ABB RAPID module: pyramid_without_orientation.mod

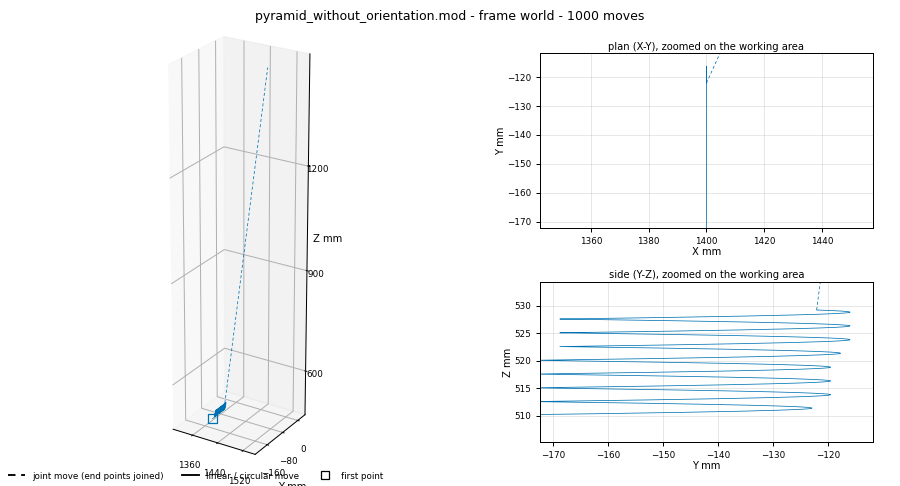
[picture p0: tool path of pyramid_without_orientation.mod in frame world, 1000 of 1000 moves have a stored position in this frame; points joined in program order, loops and branches not executed]
MODULE MainModule
    VAR string program_name:= "ProtoSocketSimulation"; !MODIFIQUE COM O NOME DO PROGRAMA ATUAL!!!!!

    VAR string received_string;
    VAR string message;
    VAR intnum timeint:=0;
    VAR intnum i:=0;
    VAR socketdev socket1;
    VAR string strTemp;
    VAR robtarget actual_pos;
    VAR intnum state;

	TASK PERS tooldata TTW5500_1:=[TRUE,[[32.1099,-0.389434,387.111],[1,0,0,0]],[1,[0,0,100],[1,0,0,0],0,0,0]];
	PERS wobjdata wobj1:=[ FALSE,TRUE,"",[[1400.0000,11.3000,510.0000],[1,0,0,0]],[[0,0,0],[1,0,0,0] ] ];

	CONST robtarget p0:=[[1455.38,0.95,1463.94],[0.707633,-0.000297139,0.70658,0.00010484],[0,0,-1,1],[9E+09,0,0,9E+09,9E+09,9E+09]];
	CONST robtarget p1:=[[0.0000,-194.9500,0.1000],[0.0000,-0.3947,0.9188,0.0000],[-1,0,-1,0],[9E+09,0.0000,0.0000,9E+09,9E+09,9E+09]];
	CONST robtarget p2:=[[0.0000,-193.5108,0.1185],[0.0000,-0.3915,0.9202,0.0000],[-1,0,-1,0],[9E+09,0.0000,-0.4058,9E+09,9E+09,9E+09]];
	CONST robtarget p3:=[[0.0000,-192.0814,0.1370],[0.0000,-0.3882,0.9216,0.0000],[-1,0,-1,0],[9E+09,0.0000,-0.8176,9E+09,9E+09,9E+09]];
	CONST robtarget p4:=[[0.0000,-190.6621,0.1556],[0.0000,-0.3848,0.9230,0.0000],[-1,0,-1,0],[9E+09,0.0000,-1.2355,9E+09,9E+09,9E+09]];
	CONST robtarget p5:=[[0.0000,-189.2531,0.1741],[0.0000,-0.3814,0.9244,0.0000],[-1,0,-1,0],[9E+09,0.0000,-1.6597,9E+09,9E+09,9E+09]];
	CONST robtarget p6:=[[0.0000,-187.8546,0.1926],[0.0000,-0.3779,0.9258,0.0000],[-1,0,-1,0],[9E+09,0.0000,-2.0903,9E+09,9E+09,9E+09]];
	CONST robtarget p7:=[[0.0000,-186.4669,0.2111],[0.0000,-0.3744,0.9273,0.0000],[-1,0,-1,0],[9E+09,0.0000,-2.5273,9E+09,9E+09,9E+09]];
	CONST robtarget p8:=[[0.0000,-185.0902,0.2296],[0.0000,-0.3708,0.9287,0.0000],[-1,0,-1,0],[9E+09,0.0000,-2.9708,9E+09,9E+09,9E+09]];
	CONST robtarget p9:=[[0.0000,-183.7248,0.2481],[0.0000,-0.3671,0.9302,0.0000],[-1,0,-1,0],[9E+09,0.0000,-3.4209,9E+09,9E+09,9E+09]];
	CONST robtarget p10:=[[0.0000,-182.3708,0.2667],[0.0000,-0.3634,0.9316,0.0000],[-1,0,-1,0],[9E+09,0.0000,-3.8777,9E+09,9E+09,9E+09]];
	CONST robtarget p11:=[[0.0000,-181.0287,0.2852],[0.0000,-0.3597,0.9331,0.0000],[-1,0,-1,0],[9E+09,0.0000,-4.3414,9E+09,9E+09,9E+09]];
	CONST robtarget p12:=[[0.0000,-179.6985,0.3037],[0.0000,-0.3558,0.9346,0.0000],[-1,0,-1,0],[9E+09,0.0000,-4.8119,9E+09,9E+09,9E+09]];
	CONST robtarget p13:=[[0.0000,-178.3807,0.3222],[0.0000,-0.3519,0.9360,0.0000],[-1,0,-1,0],[9E+09,0.0000,-5.2895,9E+09,9E+09,9E+09]];
	CONST robtarget p14:=[[0.0000,-177.0755,0.3407],[0.0000,-0.3480,0.9375,0.0000],[-1,0,-1,0],[9E+09,0.0000,-5.7741,9E+09,9E+09,9E+09]];
	CONST robtarget p15:=[[0.0000,-175.7830,0.3593],[0.0000,-0.3439,0.9390,0.0000],[-1,0,-1,0],[9E+09,0.0000,-6.2658,9E+09,9E+09,9E+09]];
	CONST robtarget p16:=[[0.0000,-174.5038,0.3778],[0.0000,-0.3398,0.9405,0.0000],[-1,0,-1,0],[9E+09,0.0000,-6.7648,9E+09,9E+09,9E+09]];
	CONST robtarget p17:=[[0.0000,-173.2379,0.3963],[0.0000,-0.3357,0.9420,0.0000],[-1,0,-1,0],[9E+09,0.0000,-7.2712,9E+09,9E+09,9E+09]];
	CONST robtarget p18:=[[0.0000,-171.9858,0.4148],[0.0000,-0.3315,0.9435,0.0000],[-1,0,-1,0],[9E+09,0.0000,-7.7849,9E+09,9E+09,9E+09]];
	CONST robtarget p19:=[[0.0000,-170.7478,0.4333],[0.0000,-0.3272,0.9450,0.0000],[-1,0,-1,0],[9E+09,0.0000,-8.3062,9E+09,9E+09,9E+09]];
	CONST robtarget p20:=[[0.0000,-169.5240,0.4519],[0.0000,-0.3228,0.9465,0.0000],[-1,0,-1,0],[9E+09,0.0000,-8.8350,9E+09,9E+09,9E+09]];
	CONST robtarget p21:=[[0.0000,-168.3149,0.4704],[0.0000,-0.3184,0.9480,0.0000],[-1,0,-1,0],[9E+09,0.0000,-9.3714,9E+09,9E+09,9E+09]];
	CONST robtarget p22:=[[0.0000,-167.1208,0.4889],[0.0000,-0.3139,0.9495,0.0000],[-1,0,-1,0],[9E+09,0.0000,-9.9156,9E+09,9E+09,9E+09]];
	CONST robtarget p23:=[[0.0000,-165.9420,0.5074],[0.0000,-0.3093,0.9510,0.0000],[-1,0,-1,0],[9E+09,0.0000,-10.4676,9E+09,9E+09,9E+09]];
	CONST robtarget p24:=[[0.0000,-164.7788,0.5259],[0.0000,-0.3046,0.9525,0.0000],[-1,0,-1,0],[9E+09,0.0000,-11.0274,9E+09,9E+09,9E+09]];
	CONST robtarget p25:=[[0.0000,-163.6315,0.5444],[0.0000,-0.2999,0.9540,0.0000],[-1,0,-1,0],[9E+09,0.0000,-11.5951,9E+09,9E+09,9E+09]];
	CONST robtarget p26:=[[0.0000,-162.5006,0.5630],[0.0000,-0.2951,0.9555,0.0000],[-1,0,-1,0],[9E+09,0.0000,-12.1707,9E+09,9E+09,9E+09]];
	CONST robtarget p27:=[[0.0000,-161.3862,0.5815],[0.0000,-0.2902,0.9570,0.0000],[-1,0,-1,0],[9E+09,0.0000,-12.7544,9E+09,9E+09,9E+09]];
	CONST robtarget p28:=[[0.0000,-160.2889,0.6000],[0.0000,-0.2853,0.9584,0.0000],[-1,0,-1,0],[9E+09,0.0000,-13.3461,9E+09,9E+09,9E+09]];
	CONST robtarget p29:=[[0.0000,-159.2088,0.6185],[0.0000,-0.2803,0.9599,0.0000],[-1,0,-1,0],[9E+09,0.0000,-13.9460,9E+09,9E+09,9E+09]];
	CONST robtarget p30:=[[0.0000,-158.1465,0.6370],[0.0000,-0.2752,0.9614,0.0000],[-1,0,-1,0],[9E+09,0.0000,-14.5539,9E+09,9E+09,9E+09]];
	CONST robtarget p31:=[[0.0000,-157.1022,0.6556],[0.0000,-0.2700,0.9629,0.0000],[-1,0,-1,0],[9E+09,0.0000,-15.1700,9E+09,9E+09,9E+09]];
	CONST robtarget p32:=[[0.0000,-156.0763,0.6741],[0.0000,-0.2648,0.9643,0.0000],[-1,0,-1,0],[9E+09,0.0000,-15.7943,9E+09,9E+09,9E+09]];
	CONST robtarget p33:=[[0.0000,-155.0692,0.6926],[0.0000,-0.2594,0.9658,0.0000],[-1,0,-1,0],[9E+09,0.0000,-16.4267,9E+09,9E+09,9E+09]];
	CONST robtarget p34:=[[0.0000,-154.0812,0.7111],[0.0000,-0.2540,0.9672,0.0000],[-1,0,-1,0],[9E+09,0.0000,-17.0674,9E+09,9E+09,9E+09]];
	CONST robtarget p35:=[[0.0000,-153.1128,0.7296],[0.0000,-0.2486,0.9686,0.0000],[-1,0,-1,0],[9E+09,0.0000,-17.7162,9E+09,9E+09,9E+09]];
	CONST robtarget p36:=[[0.0000,-152.1642,0.7481],[0.0000,-0.2430,0.9700,0.0000],[-1,0,-1,0],[9E+09,0.0000,-18.3732,9E+09,9E+09,9E+09]];
	CONST robtarget p37:=[[0.0000,-151.2359,0.7667],[0.0000,-0.2374,0.9714,0.0000],[-1,0,-1,0],[9E+09,0.0000,-19.0384,9E+09,9E+09,9E+09]];
	CONST robtarget p38:=[[0.0000,-150.3282,0.7852],[0.0000,-0.2316,0.9728,0.0000],[-1,0,-1,0],[9E+09,0.0000,-19.7117,9E+09,9E+09,9E+09]];
	CONST robtarget p39:=[[0.0000,-149.4415,0.8037],[0.0000,-0.2259,0.9742,0.0000],[-1,0,-1,0],[9E+09,0.0000,-20.3930,9E+09,9E+09,9E+09]];
	CONST robtarget p40:=[[0.0000,-148.5762,0.8222],[0.0000,-0.2200,0.9755,0.0000],[-1,0,-1,0],[9E+09,0.0000,-21.0824,9E+09,9E+09,9E+09]];
	CONST robtarget p41:=[[0.0000,-147.7327,0.8407],[0.0000,-0.2141,0.9768,0.0000],[-1,0,-1,0],[9E+09,0.0000,-21.7798,9E+09,9E+09,9E+09]];
	CONST robtarget p42:=[[0.0000,-146.9113,0.8593],[0.0000,-0.2080,0.9781,0.0000],[-1,0,-1,0],[9E+09,0.0000,-22.4851,9E+09,9E+09,9E+09]];
	CONST robtarget p43:=[[0.0000,-146.1124,0.8778],[0.0000,-0.2019,0.9794,0.0000],[-1,0,-1,0],[9E+09,0.0000,-23.1982,9E+09,9E+09,9E+09]];
	CONST robtarget p44:=[[0.0000,-145.3364,0.8963],[0.0000,-0.1958,0.9806,0.0000],[-1,0,-1,0],[9E+09,0.0000,-23.9190,9E+09,9E+09,9E+09]];
	CONST robtarget p45:=[[0.0000,-144.5836,0.9148],[0.0000,-0.1895,0.9819,0.0000],[-1,0,-1,0],[9E+09,0.0000,-24.6475,9E+09,9E+09,9E+09]];
	CONST robtarget p46:=[[0.0000,-143.8545,0.9333],[0.0000,-0.1832,0.9831,0.0000],[-1,0,-1,0],[9E+09,0.0000,-25.3834,9E+09,9E+09,9E+09]];
	CONST robtarget p47:=[[0.0000,-143.1493,0.9519],[0.0000,-0.1769,0.9842,0.0000],[-1,0,-1,0],[9E+09,0.0000,-26.1268,9E+09,9E+09,9E+09]];
	CONST robtarget p48:=[[0.0000,-142.4685,0.9704],[0.0000,-0.1704,0.9854,0.0000],[-1,0,-1,0],[9E+09,0.0000,-26.8773,9E+09,9E+09,9E+09]];
	CONST robtarget p49:=[[0.0000,-141.8123,0.9889],[0.0000,-0.1639,0.9865,0.0000],[-1,0,-1,0],[9E+09,0.0000,-27.6350,9E+09,9E+09,9E+09]];
	CONST robtarget p50:=[[0.0000,-141.1812,1.0074],[0.0000,-0.1573,0.9876,0.0000],[-1,0,-1,0],[9E+09,0.0000,-28.3995,9E+09,9E+09,9E+09]];
	CONST robtarget p51:=[[0.0000,-140.5754,1.0259],[0.0000,-0.1507,0.9886,0.0000],[-1,0,-1,0],[9E+09,0.0000,-29.1708,9E+09,9E+09,9E+09]];
	CONST robtarget p52:=[[0.0000,-139.9953,1.0444],[0.0000,-0.1439,0.9896,0.0000],[-1,0,-1,0],[9E+09,0.0000,-29.9486,9E+09,9E+09,9E+09]];
	CONST robtarget p53:=[[0.0000,-139.4412,1.0630],[0.0000,-0.1372,0.9905,0.0000],[-1,0,-1,0],[9E+09,0.0000,-30.7328,9E+09,9E+09,9E+09]];
	CONST robtarget p54:=[[0.0000,-138.9135,1.0815],[0.0000,-0.1303,0.9915,0.0000],[-1,0,-1,0],[9E+09,0.0000,-31.5230,9E+09,9E+09,9E+09]];
	CONST robtarget p55:=[[0.0000,-138.4124,1.1000],[0.0000,-0.1234,0.9924,0.0000],[-1,0,-1,0],[9E+09,0.0000,-32.3191,9E+09,9E+09,9E+09]];
	CONST robtarget p56:=[[0.0000,-137.9381,1.1185],[0.0000,-0.1165,0.9932,0.0000],[-1,0,-1,0],[9E+09,0.0000,-33.1209,9E+09,9E+09,9E+09]];
	CONST robtarget p57:=[[0.0000,-137.4911,1.1370],[0.0000,-0.1095,0.9940,0.0000],[-1,0,-1,0],[9E+09,0.0000,-33.9280,9E+09,9E+09,9E+09]];
	CONST robtarget p58:=[[0.0000,-137.0716,1.1556],[0.0000,-0.1024,0.9947,0.0000],[-1,0,-1,0],[9E+09,0.0000,-34.7402,9E+09,9E+09,9E+09]];
	CONST robtarget p59:=[[0.0000,-136.6797,1.1741],[0.0000,-0.0953,0.9954,0.0000],[-1,0,-1,0],[9E+09,0.0000,-35.5573,9E+09,9E+09,9E+09]];
	CONST robtarget p60:=[[0.0000,-136.3158,1.1926],[0.0000,-0.0882,0.9961,0.0000],[-1,0,-1,0],[9E+09,0.0000,-36.3788,9E+09,9E+09,9E+09]];
	CONST robtarget p61:=[[0.0000,-135.9801,1.2111],[0.0000,-0.0810,0.9967,0.0000],[-1,0,-1,0],[9E+09,0.0000,-37.2046,9E+09,9E+09,9E+09]];
	CONST robtarget p62:=[[0.0000,-135.6728,1.2296],[0.0000,-0.0738,0.9973,0.0000],[-1,0,-1,0],[9E+09,0.0000,-38.0344,9E+09,9E+09,9E+09]];
	CONST robtarget p63:=[[0.0000,-135.3940,1.2481],[0.0000,-0.0666,0.9978,0.0000],[-1,0,-1,0],[9E+09,0.0000,-38.8677,9E+09,9E+09,9E+09]];
	CONST robtarget p64:=[[0.0000,-135.1440,1.2667],[0.0000,-0.0593,0.9982,0.0000],[-1,0,-1,0],[9E+09,0.0000,-39.7042,9E+09,9E+09,9E+09]];
	CONST robtarget p65:=[[0.0000,-134.9229,1.2852],[0.0000,-0.0520,0.9986,0.0000],[-1,0,-1,0],[9E+09,0.0000,-40.5437,9E+09,9E+09,9E+09]];
	CONST robtarget p66:=[[0.0000,-134.7309,1.3037],[0.0000,-0.0446,0.9990,0.0000],[-1,0,-1,0],[9E+09,0.0000,-41.3858,9E+09,9E+09,9E+09]];
	CONST robtarget p67:=[[0.0000,-134.5680,1.3222],[0.0000,-0.0373,0.9993,0.0000],[-1,0,-1,0],[9E+09,0.0000,-42.2301,9E+09,9E+09,9E+09]];
	CONST robtarget p68:=[[0.0000,-134.4344,1.3407],[0.0000,-0.0299,0.9996,0.0000],[-1,0,-1,0],[9E+09,0.0000,-43.0762,9E+09,9E+09,9E+09]];
	CONST robtarget p69:=[[0.0000,-134.3302,1.3593],[0.0000,-0.0225,0.9997,0.0000],[-1,0,-1,0],[9E+09,0.0000,-43.9239,9E+09,9E+09,9E+09]];
	CONST robtarget p70:=[[0.0000,-134.2555,1.3778],[0.0000,-0.0151,0.9999,0.0000],[-1,0,-1,0],[9E+09,0.0000,-44.7727,9E+09,9E+09,9E+09]];
	CONST robtarget p71:=[[0.0000,-134.2102,1.3963],[0.0000,-0.0077,1.0000,0.0000],[-1,0,-1,0],[9E+09,0.0000,-45.6222,9E+09,9E+09,9E+09]];
	CONST robtarget p72:=[[0.0000,-134.1945,1.4148],[0.0000,-0.0002,1.0000,0.0000],[-1,0,-1,0],[9E+09,0.0000,-46.4721,9E+09,9E+09,9E+09]];
	CONST robtarget p73:=[[0.0000,-134.2083,1.4333],[0.0000,-0.0072,-1.0000,0.0000],[-1,0,-1,0],[9E+09,0.0000,-47.3221,9E+09,9E+09,9E+09]];
	CONST robtarget p74:=[[0.0000,-134.2516,1.4519],[0.0000,-0.0146,-0.9999,0.0000],[-1,0,-1,0],[9E+09,0.0000,-48.1716,9E+09,9E+09,9E+09]];
	CONST robtarget p75:=[[0.0000,-134.3244,1.4704],[0.0000,-0.0220,-0.9998,0.0000],[-1,0,-1,0],[9E+09,0.0000,-49.0205,9E+09,9E+09,9E+09]];
	CONST robtarget p76:=[[0.0000,-134.4267,1.4889],[0.0000,-0.0294,-0.9996,0.0000],[-1,0,-1,0],[9E+09,0.0000,-49.8682,9E+09,9E+09,9E+09]];
	CONST robtarget p77:=[[0.0000,-134.5583,1.5074],[0.0000,-0.0368,-0.9993,0.0000],[-1,0,-1,0],[9E+09,0.0000,-50.7145,9E+09,9E+09,9E+09]];
	CONST robtarget p78:=[[0.0000,-134.7192,1.5259],[0.0000,-0.0441,-0.9990,0.0000],[-1,0,-1,0],[9E+09,0.0000,-51.5589,9E+09,9E+09,9E+09]];
	CONST robtarget p79:=[[0.0000,-134.9094,1.5444],[0.0000,-0.0515,-0.9987,0.0000],[-1,0,-1,0],[9E+09,0.0000,-52.4011,9E+09,9E+09,9E+09]];
	CONST robtarget p80:=[[0.0000,-135.1285,1.5630],[0.0000,-0.0588,-0.9983,0.0000],[-1,0,-1,0],[9E+09,0.0000,-53.2408,9E+09,9E+09,9E+09]];
	CONST robtarget p81:=[[0.0000,-135.3767,1.5815],[0.0000,-0.0661,-0.9978,0.0000],[-1,0,-1,0],[9E+09,0.0000,-54.0776,9E+09,9E+09,9E+09]];
	CONST robtarget p82:=[[0.0000,-135.6535,1.6000],[0.0000,-0.0733,-0.9973,0.0000],[-1,0,-1,0],[9E+09,0.0000,-54.9111,9E+09,9E+09,9E+09]];
	CONST robtarget p83:=[[0.0000,-135.9590,1.6185],[0.0000,-0.0806,-0.9968,0.0000],[-1,0,-1,0],[9E+09,0.0000,-55.7411,9E+09,9E+09,9E+09]];
	CONST robtarget p84:=[[0.0000,-136.2929,1.6370],[0.0000,-0.0877,-0.9961,0.0000],[-1,0,-1,0],[9E+09,0.0000,-56.5671,9E+09,9E+09,9E+09]];
	CONST robtarget p85:=[[0.0000,-136.6549,1.6556],[0.0000,-0.0949,-0.9955,0.0000],[-1,0,-1,0],[9E+09,0.0000,-57.3890,9E+09,9E+09,9E+09]];
	CONST robtarget p86:=[[0.0000,-137.0449,1.6741],[0.0000,-0.1020,-0.9948,0.0000],[-1,0,-1,0],[9E+09,0.0000,-58.2064,9E+09,9E+09,9E+09]];
	CONST robtarget p87:=[[0.0000,-137.4627,1.6926],[0.0000,-0.1090,-0.9940,0.0000],[-1,0,-1,0],[9E+09,0.0000,-59.0189,9E+09,9E+09,9E+09]];
	CONST robtarget p88:=[[0.0000,-137.9079,1.7111],[0.0000,-0.1160,-0.9932,0.0000],[-1,0,-1,0],[9E+09,0.0000,-59.8264,9E+09,9E+09,9E+09]];
	CONST robtarget p89:=[[0.0000,-138.3803,1.7296],[0.0000,-0.1230,-0.9924,0.0000],[-1,0,-1,0],[9E+09,0.0000,-60.6285,9E+09,9E+09,9E+09]];
	CONST robtarget p90:=[[0.0000,-138.8797,1.7481],[0.0000,-0.1299,-0.9915,0.0000],[-1,0,-1,0],[9E+09,0.0000,-61.4250,9E+09,9E+09,9E+09]];
	CONST robtarget p91:=[[0.0000,-139.4057,1.7667],[0.0000,-0.1367,-0.9906,0.0000],[-1,0,-1,0],[9E+09,0.0000,-62.2156,9E+09,9E+09,9E+09]];
	CONST robtarget p92:=[[0.0000,-139.9580,1.7852],[0.0000,-0.1435,-0.9897,0.0000],[-1,0,-1,0],[9E+09,0.0000,-63.0002,9E+09,9E+09,9E+09]];
	CONST robtarget p93:=[[0.0000,-140.5364,1.8037],[0.0000,-0.1502,-0.9887,0.0000],[-1,0,-1,0],[9E+09,0.0000,-63.7784,9E+09,9E+09,9E+09]];
	CONST robtarget p94:=[[0.0000,-141.1405,1.8222],[0.0000,-0.1569,-0.9876,0.0000],[-1,0,-1,0],[9E+09,0.0000,-64.5501,9E+09,9E+09,9E+09]];
	CONST robtarget p95:=[[0.0000,-141.7700,1.8407],[0.0000,-0.1635,-0.9866,0.0000],[-1,0,-1,0],[9E+09,0.0000,-65.3151,9E+09,9E+09,9E+09]];
	CONST robtarget p96:=[[0.0000,-142.4245,1.8593],[0.0000,-0.1700,-0.9854,0.0000],[-1,0,-1,0],[9E+09,0.0000,-66.0732,9E+09,9E+09,9E+09]];
	CONST robtarget p97:=[[0.0000,-143.1037,1.8778],[0.0000,-0.1764,-0.9843,0.0000],[-1,0,-1,0],[9E+09,0.0000,-66.8242,9E+09,9E+09,9E+09]];
	CONST robtarget p98:=[[0.0000,-143.8073,1.8963],[0.0000,-0.1828,-0.9831,0.0000],[-1,0,-1,0],[9E+09,0.0000,-67.5681,9E+09,9E+09,9E+09]];
	CONST robtarget p99:=[[0.0000,-144.5349,1.9148],[0.0000,-0.1891,-0.9820,0.0000],[-1,0,-1,0],[9E+09,0.0000,-68.3045,9E+09,9E+09,9E+09]];
	CONST robtarget p100:=[[0.0000,-145.2861,1.9333],[0.0000,-0.1954,-0.9807,0.0000],[-1,0,-1,0],[9E+09,0.0000,-69.0335,9E+09,9E+09,9E+09]];
	CONST robtarget p101:=[[0.0000,-146.0606,1.9519],[0.0000,-0.2015,-0.9795,0.0000],[-1,0,-1,0],[9E+09,0.0000,-69.7548,9E+09,9E+09,9E+09]];
	CONST robtarget p102:=[[0.0000,-146.8580,1.9704],[0.0000,-0.2076,-0.9782,0.0000],[-1,0,-1,0],[9E+09,0.0000,-70.4684,9E+09,9E+09,9E+09]];
	CONST robtarget p103:=[[0.0000,-147.6779,1.9889],[0.0000,-0.2137,-0.9769,0.0000],[-1,0,-1,0],[9E+09,0.0000,-71.1742,9E+09,9E+09,9E+09]];
	CONST robtarget p104:=[[0.0000,-148.5200,2.0074],[0.0000,-0.2196,-0.9756,0.0000],[-1,0,-1,0],[9E+09,0.0000,-71.8721,9E+09,9E+09,9E+09]];
	CONST robtarget p105:=[[0.0000,-149.3839,2.0259],[0.0000,-0.2255,-0.9742,0.0000],[-1,0,-1,0],[9E+09,0.0000,-72.5620,9E+09,9E+09,9E+09]];
	CONST robtarget p106:=[[0.0000,-150.2692,2.0444],[0.0000,-0.2313,-0.9729,0.0000],[-1,0,-1,0],[9E+09,0.0000,-73.2439,9E+09,9E+09,9E+09]];
	CONST robtarget p107:=[[0.0000,-151.1755,2.0630],[0.0000,-0.2370,-0.9715,0.0000],[-1,0,-1,0],[9E+09,0.0000,-73.9178,9E+09,9E+09,9E+09]];
	CONST robtarget p108:=[[0.0000,-152.1025,2.0815],[0.0000,-0.2426,-0.9701,0.0000],[-1,0,-1,0],[9E+09,0.0000,-74.5835,9E+09,9E+09,9E+09]];
	CONST robtarget p109:=[[0.0000,-153.0497,2.1000],[0.0000,-0.2482,-0.9687,0.0000],[-1,0,-1,0],[9E+09,0.0000,-75.2410,9E+09,9E+09,9E+09]];
	CONST robtarget p110:=[[0.0000,-154.0169,2.1185],[0.0000,-0.2537,-0.9673,0.0000],[-1,0,-1,0],[9E+09,0.0000,-75.8904,9E+09,9E+09,9E+09]];
	CONST robtarget p111:=[[0.0000,-155.0036,2.1370],[0.0000,-0.2591,-0.9659,0.0000],[-1,0,-1,0],[9E+09,0.0000,-76.5316,9E+09,9E+09,9E+09]];
	CONST robtarget p112:=[[0.0000,-156.0095,2.1556],[0.0000,-0.2644,-0.9644,0.0000],[-1,0,-1,0],[9E+09,0.0000,-77.1646,9E+09,9E+09,9E+09]];
	CONST robtarget p113:=[[0.0000,-157.0341,2.1741],[0.0000,-0.2697,-0.9630,0.0000],[-1,0,-1,0],[9E+09,0.0000,-77.7894,9E+09,9E+09,9E+09]];
	CONST robtarget p114:=[[0.0000,-158.0772,2.1926],[0.0000,-0.2748,-0.9615,0.0000],[-1,0,-1,0],[9E+09,0.0000,-78.4060,9E+09,9E+09,9E+09]];
	CONST robtarget p115:=[[0.0000,-159.1384,2.2111],[0.0000,-0.2799,-0.9600,0.0000],[-1,0,-1,0],[9E+09,0.0000,-79.0145,9E+09,9E+09,9E+09]];
	CONST robtarget p116:=[[0.0000,-160.2172,2.2296],[0.0000,-0.2850,-0.9585,0.0000],[-1,0,-1,0],[9E+09,0.0000,-79.6148,9E+09,9E+09,9E+09]];
	CONST robtarget p117:=[[0.0000,-161.3135,2.2481],[0.0000,-0.2899,-0.9570,0.0000],[-1,0,-1,0],[9E+09,0.0000,-80.2071,9E+09,9E+09,9E+09]];
	CONST robtarget p118:=[[0.0000,-162.4267,2.2667],[0.0000,-0.2948,-0.9556,0.0000],[-1,0,-1,0],[9E+09,0.0000,-80.7913,9E+09,9E+09,9E+09]];
	CONST robtarget p119:=[[0.0000,-163.5566,2.2852],[0.0000,-0.2996,-0.9541,0.0000],[-1,0,-1,0],[9E+09,0.0000,-81.3675,9E+09,9E+09,9E+09]];
	CONST robtarget p120:=[[0.0000,-164.7028,2.3037],[0.0000,-0.3043,-0.9526,0.0000],[-1,0,-1,0],[9E+09,0.0000,-81.9357,9E+09,9E+09,9E+09]];
	CONST robtarget p121:=[[0.0000,-165.8649,2.3222],[0.0000,-0.3090,-0.9511,0.0000],[-1,0,-1,0],[9E+09,0.0000,-82.4960,9E+09,9E+09,9E+09]];
	CONST robtarget p122:=[[0.0000,-167.0428,2.3407],[0.0000,-0.3136,-0.9496,0.0000],[-1,0,-1,0],[9E+09,0.0000,-83.0485,9E+09,9E+09,9E+09]];
	CONST robtarget p123:=[[0.0000,-168.2359,2.3593],[0.0000,-0.3181,-0.9481,0.0000],[-1,0,-1,0],[9E+09,0.0000,-83.5932,9E+09,9E+09,9E+09]];
	CONST robtarget p124:=[[0.0000,-169.4440,2.3778],[0.0000,-0.3225,-0.9466,0.0000],[-1,0,-1,0],[9E+09,0.0000,-84.1301,9E+09,9E+09,9E+09]];
	CONST robtarget p125:=[[0.0000,-170.6668,2.3963],[0.0000,-0.3269,-0.9451,0.0000],[-1,0,-1,0],[9E+09,0.0000,-84.6595,9E+09,9E+09,9E+09]];
	CONST robtarget p126:=[[0.0000,-171.9039,2.4148],[0.0000,-0.3312,-0.9436,0.0000],[-1,0,-1,0],[9E+09,0.0000,-85.1812,9E+09,9E+09,9E+09]];
	CONST robtarget p127:=[[0.0000,-173.1551,2.4333],[0.0000,-0.3354,-0.9421,0.0000],[-1,0,-1,0],[9E+09,0.0000,-85.6954,9E+09,9E+09,9E+09]];
	CONST robtarget p128:=[[0.0000,-174.4200,2.4519],[0.0000,-0.3396,-0.9406,0.0000],[-1,0,-1,0],[9E+09,0.0000,-86.2023,9E+09,9E+09,9E+09]];
	CONST robtarget p129:=[[0.0000,-175.6984,2.4704],[0.0000,-0.3437,-0.9391,0.0000],[-1,0,-1,0],[9E+09,0.0000,-86.7018,9E+09,9E+09,9E+09]];
	CONST robtarget p130:=[[0.0000,-176.9900,2.4889],[0.0000,-0.3477,-0.9376,0.0000],[-1,0,-1,0],[9E+09,0.0000,-87.1940,9E+09,9E+09,9E+09]];
	CONST robtarget p131:=[[0.0000,-178.2944,2.5074],[0.0000,-0.3517,-0.9361,0.0000],[-1,0,-1,0],[9E+09,0.0000,-87.6791,9E+09,9E+09,9E+09]];
	CONST robtarget p132:=[[0.0000,-179.6114,2.5259],[0.0000,-0.3556,-0.9346,0.0000],[-1,0,-1,0],[9E+09,0.0000,-88.1571,9E+09,9E+09,9E+09]];
	CONST robtarget p133:=[[0.0000,-180.9408,2.5444],[0.0000,-0.3594,-0.9332,0.0000],[-1,0,-1,0],[9E+09,0.0000,-88.6280,9E+09,9E+09,9E+09]];
	CONST robtarget p134:=[[0.0000,-182.2821,2.5630],[0.0000,-0.3632,-0.9317,0.0000],[-1,0,-1,0],[9E+09,0.0000,-89.0921,9E+09,9E+09,9E+09]];
	CONST robtarget p135:=[[0.0000,-183.6353,2.5815],[0.0000,-0.3669,-0.9303,0.0000],[-1,0,-1,0],[9E+09,0.0000,-89.5494,9E+09,9E+09,9E+09]];
	CONST robtarget p136:=[[0.0000,-185.0000,2.6000],[0.0000,-0.3827,0.9239,0.0000],[-1,0,-1,0],[9E+09,0.0000,-90.0000,9E+09,9E+09,9E+09]];
	CONST robtarget p137:=[[0.0000,-183.5932,2.6191],[0.0000,-0.3791,0.9253,0.0000],[-1,0,-1,0],[9E+09,0.0000,-90.4407,9E+09,9E+09,9E+09]];
	CONST robtarget p138:=[[0.0000,-182.1975,2.6382],[0.0000,-0.3755,0.9268,0.0000],[-1,0,-1,0],[9E+09,0.0000,-90.8882,9E+09,9E+09,9E+09]];
	CONST robtarget p139:=[[0.0000,-180.8130,2.6573],[0.0000,-0.3718,0.9283,0.0000],[-1,0,-1,0],[9E+09,0.0000,-91.3426,9E+09,9E+09,9E+09]];
	CONST robtarget p140:=[[0.0000,-179.4401,2.6763],[0.0000,-0.3681,0.9298,0.0000],[-1,0,-1,0],[9E+09,0.0000,-91.8040,9E+09,9E+09,9E+09]];
	CONST robtarget p141:=[[0.0000,-178.0790,2.6954],[0.0000,-0.3643,0.9313,0.0000],[-1,0,-1,0],[9E+09,0.0000,-92.2724,9E+09,9E+09,9E+09]];
	CONST robtarget p142:=[[0.0000,-176.7300,2.7145],[0.0000,-0.3604,0.9328,0.0000],[-1,0,-1,0],[9E+09,0.0000,-92.7481,9E+09,9E+09,9E+09]];
	CONST robtarget p143:=[[0.0000,-175.3933,2.7336],[0.0000,-0.3565,0.9343,0.0000],[-1,0,-1,0],[9E+09,0.0000,-93.2310,9E+09,9E+09,9E+09]];
	CONST robtarget p144:=[[0.0000,-174.0693,2.7527],[0.0000,-0.3525,0.9358,0.0000],[-1,0,-1,0],[9E+09,0.0000,-93.7213,9E+09,9E+09,9E+09]];
	CONST robtarget p145:=[[0.0000,-172.7582,2.7718],[0.0000,-0.3484,0.9373,0.0000],[-1,0,-1,0],[9E+09,0.0000,-94.2191,9E+09,9E+09,9E+09]];
	CONST robtarget p146:=[[0.0000,-171.4604,2.7908],[0.0000,-0.3443,0.9389,0.0000],[-1,0,-1,0],[9E+09,0.0000,-94.7245,9E+09,9E+09,9E+09]];
	CONST robtarget p147:=[[0.0000,-170.1762,2.8099],[0.0000,-0.3401,0.9404,0.0000],[-1,0,-1,0],[9E+09,0.0000,-95.2375,9E+09,9E+09,9E+09]];
	CONST robtarget p148:=[[0.0000,-168.9057,2.8290],[0.0000,-0.3358,0.9419,0.0000],[-1,0,-1,0],[9E+09,0.0000,-95.7583,9E+09,9E+09,9E+09]];
	CONST robtarget p149:=[[0.0000,-167.6495,2.8481],[0.0000,-0.3314,0.9435,0.0000],[-1,0,-1,0],[9E+09,0.0000,-96.2869,9E+09,9E+09,9E+09]];
	CONST robtarget p150:=[[0.0000,-166.4077,2.8672],[0.0000,-0.3270,0.9450,0.0000],[-1,0,-1,0],[9E+09,0.0000,-96.8235,9E+09,9E+09,9E+09]];
	CONST robtarget p151:=[[0.0000,-165.1807,2.8863],[0.0000,-0.3225,0.9466,0.0000],[-1,0,-1,0],[9E+09,0.0000,-97.3681,9E+09,9E+09,9E+09]];
	CONST robtarget p152:=[[0.0000,-163.9689,2.9053],[0.0000,-0.3180,0.9481,0.0000],[-1,0,-1,0],[9E+09,0.0000,-97.9207,9E+09,9E+09,9E+09]];
	CONST robtarget p153:=[[0.0000,-162.7726,2.9244],[0.0000,-0.3133,0.9496,0.0000],[-1,0,-1,0],[9E+09,0.0000,-98.4816,9E+09,9E+09,9E+09]];
	CONST robtarget p154:=[[0.0000,-161.5921,2.9435],[0.0000,-0.3086,0.9512,0.0000],[-1,0,-1,0],[9E+09,0.0000,-99.0507,9E+09,9E+09,9E+09]];
	CONST robtarget p155:=[[0.0000,-160.4277,2.9626],[0.0000,-0.3038,0.9527,0.0000],[-1,0,-1,0],[9E+09,0.0000,-99.6282,9E+09,9E+09,9E+09]];
	CONST robtarget p156:=[[0.0000,-159.2799,2.9817],[0.0000,-0.2989,0.9543,0.0000],[-1,0,-1,0],[9E+09,0.0000,-100.2140,9E+09,9E+09,9E+09]];
	CONST robtarget p157:=[[0.0000,-158.1490,3.0008],[0.0000,-0.2940,0.9558,0.0000],[-1,0,-1,0],[9E+09,0.0000,-100.8082,9E+09,9E+09,9E+09]];
	CONST robtarget p158:=[[0.0000,-157.0354,3.0198],[0.0000,-0.2889,0.9573,0.0000],[-1,0,-1,0],[9E+09,0.0000,-101.4110,9E+09,9E+09,9E+09]];
	CONST robtarget p159:=[[0.0000,-155.9394,3.0389],[0.0000,-0.2838,0.9589,0.0000],[-1,0,-1,0],[9E+09,0.0000,-102.0223,9E+09,9E+09,9E+09]];
	CONST robtarget p160:=[[0.0000,-154.8613,3.0580],[0.0000,-0.2786,0.9604,0.0000],[-1,0,-1,0],[9E+09,0.0000,-102.6422,9E+09,9E+09,9E+09]];
	CONST robtarget p161:=[[0.0000,-153.8017,3.0771],[0.0000,-0.2734,0.9619,0.0000],[-1,0,-1,0],[9E+09,0.0000,-103.2706,9E+09,9E+09,9E+09]];
	CONST robtarget p162:=[[0.0000,-152.7608,3.0962],[0.0000,-0.2680,0.9634,0.0000],[-1,0,-1,0],[9E+09,0.0000,-103.9078,9E+09,9E+09,9E+09]];
	CONST robtarget p163:=[[0.0000,-151.7391,3.1153],[0.0000,-0.2626,0.9649,0.0000],[-1,0,-1,0],[9E+09,0.0000,-104.5536,9E+09,9E+09,9E+09]];
	CONST robtarget p164:=[[0.0000,-150.7369,3.1344],[0.0000,-0.2571,0.9664,0.0000],[-1,0,-1,0],[9E+09,0.0000,-105.2080,9E+09,9E+09,9E+09]];
	CONST robtarget p165:=[[0.0000,-149.7546,3.1534],[0.0000,-0.2515,0.9679,0.0000],[-1,0,-1,0],[9E+09,0.0000,-105.8712,9E+09,9E+09,9E+09]];
	CONST robtarget p166:=[[0.0000,-148.7927,3.1725],[0.0000,-0.2458,0.9693,0.0000],[-1,0,-1,0],[9E+09,0.0000,-106.5430,9E+09,9E+09,9E+09]];
	CONST robtarget p167:=[[0.0000,-147.8514,3.1916],[0.0000,-0.2400,0.9708,0.0000],[-1,0,-1,0],[9E+09,0.0000,-107.2234,9E+09,9E+09,9E+09]];
	CONST robtarget p168:=[[0.0000,-146.9313,3.2107],[0.0000,-0.2342,0.9722,0.0000],[-1,0,-1,0],[9E+09,0.0000,-107.9125,9E+09,9E+09,9E+09]];
	CONST robtarget p169:=[[0.0000,-146.0327,3.2298],[0.0000,-0.2283,0.9736,0.0000],[-1,0,-1,0],[9E+09,0.0000,-108.6102,9E+09,9E+09,9E+09]];
	CONST robtarget p170:=[[0.0000,-145.1561,3.2489],[0.0000,-0.2223,0.9750,0.0000],[-1,0,-1,0],[9E+09,0.0000,-109.3164,9E+09,9E+09,9E+09]];
	CONST robtarget p171:=[[0.0000,-144.3017,3.2679],[0.0000,-0.2162,0.9764,0.0000],[-1,0,-1,0],[9E+09,0.0000,-110.0310,9E+09,9E+09,9E+09]];
	CONST robtarget p172:=[[0.0000,-143.4701,3.2870],[0.0000,-0.2100,0.9777,0.0000],[-1,0,-1,0],[9E+09,0.0000,-110.7541,9E+09,9E+09,9E+09]];
	CONST robtarget p173:=[[0.0000,-142.6615,3.3061],[0.0000,-0.2038,0.9790,0.0000],[-1,0,-1,0],[9E+09,0.0000,-111.4854,9E+09,9E+09,9E+09]];
	CONST robtarget p174:=[[0.0000,-141.8765,3.3252],[0.0000,-0.1974,0.9803,0.0000],[-1,0,-1,0],[9E+09,0.0000,-112.2250,9E+09,9E+09,9E+09]];
	CONST robtarget p175:=[[0.0000,-141.1154,3.3443],[0.0000,-0.1910,0.9816,0.0000],[-1,0,-1,0],[9E+09,0.0000,-112.9727,9E+09,9E+09,9E+09]];
	CONST robtarget p176:=[[0.0000,-140.3786,3.3634],[0.0000,-0.1846,0.9828,0.0000],[-1,0,-1,0],[9E+09,0.0000,-113.7284,9E+09,9E+09,9E+09]];
	CONST robtarget p177:=[[0.0000,-139.6664,3.3824],[0.0000,-0.1780,0.9840,0.0000],[-1,0,-1,0],[9E+09,0.0000,-114.4919,9E+09,9E+09,9E+09]];
	CONST robtarget p178:=[[0.0000,-138.9793,3.4015],[0.0000,-0.1714,0.9852,0.0000],[-1,0,-1,0],[9E+09,0.0000,-115.2631,9E+09,9E+09,9E+09]];
	CONST robtarget p179:=[[0.0000,-138.3177,3.4206],[0.0000,-0.1647,0.9863,0.0000],[-1,0,-1,0],[9E+09,0.0000,-116.0418,9E+09,9E+09,9E+09]];
	CONST robtarget p180:=[[0.0000,-137.6818,3.4397],[0.0000,-0.1579,0.9875,0.0000],[-1,0,-1,0],[9E+09,0.0000,-116.8279,9E+09,9E+09,9E+09]];
	CONST robtarget p181:=[[0.0000,-137.0721,3.4588],[0.0000,-0.1511,0.9885,0.0000],[-1,0,-1,0],[9E+09,0.0000,-117.6211,9E+09,9E+09,9E+09]];
	CONST robtarget p182:=[[0.0000,-136.4888,3.4779],[0.0000,-0.1442,0.9896,0.0000],[-1,0,-1,0],[9E+09,0.0000,-118.4212,9E+09,9E+09,9E+09]];
	CONST robtarget p183:=[[0.0000,-135.9325,3.4969],[0.0000,-0.1372,0.9905,0.0000],[-1,0,-1,0],[9E+09,0.0000,-119.2281,9E+09,9E+09,9E+09]];
	CONST robtarget p184:=[[0.0000,-135.4032,3.5160],[0.0000,-0.1302,0.9915,0.0000],[-1,0,-1,0],[9E+09,0.0000,-120.0414,9E+09,9E+09,9E+09]];
	CONST robtarget p185:=[[0.0000,-134.9015,3.5351],[0.0000,-0.1231,0.9924,0.0000],[-1,0,-1,0],[9E+09,0.0000,-120.8609,9E+09,9E+09,9E+09]];
	CONST robtarget p186:=[[0.0000,-134.4276,3.5542],[0.0000,-0.1159,0.9933,0.0000],[-1,0,-1,0],[9E+09,0.0000,-121.6864,9E+09,9E+09,9E+09]];
	CONST robtarget p187:=[[0.0000,-133.9818,3.5733],[0.0000,-0.1087,0.9941,0.0000],[-1,0,-1,0],[9E+09,0.0000,-122.5175,9E+09,9E+09,9E+09]];
	CONST robtarget p188:=[[0.0000,-133.5644,3.5924],[0.0000,-0.1015,0.9948,0.0000],[-1,0,-1,0],[9E+09,0.0000,-123.3540,9E+09,9E+09,9E+09]];
	CONST robtarget p189:=[[0.0000,-133.1756,3.6115],[0.0000,-0.0941,0.9956,0.0000],[-1,0,-1,0],[9E+09,0.0000,-124.1956,9E+09,9E+09,9E+09]];
	CONST robtarget p190:=[[0.0000,-132.8157,3.6305],[0.0000,-0.0868,0.9962,0.0000],[-1,0,-1,0],[9E+09,0.0000,-125.0419,9E+09,9E+09,9E+09]];
	CONST robtarget p191:=[[0.0000,-132.4849,3.6496],[0.0000,-0.0794,0.9968,0.0000],[-1,0,-1,0],[9E+09,0.0000,-125.8927,9E+09,9E+09,9E+09]];
	CONST robtarget p192:=[[0.0000,-132.1835,3.6687],[0.0000,-0.0720,0.9974,0.0000],[-1,0,-1,0],[9E+09,0.0000,-126.7475,9E+09,9E+09,9E+09]];
	CONST robtarget p193:=[[0.0000,-131.9116,3.6878],[0.0000,-0.0645,0.9979,0.0000],[-1,0,-1,0],[9E+09,0.0000,-127.6060,9E+09,9E+09,9E+09]];
	CONST robtarget p194:=[[0.0000,-131.6695,3.7069],[0.0000,-0.0570,0.9984,0.0000],[-1,0,-1,0],[9E+09,0.0000,-128.4679,9E+09,9E+09,9E+09]];
	CONST robtarget p195:=[[0.0000,-131.4573,3.7260],[0.0000,-0.0494,0.9988,0.0000],[-1,0,-1,0],[9E+09,0.0000,-129.3327,9E+09,9E+09,9E+09]];
	CONST robtarget p196:=[[0.0000,-131.2751,3.7450],[0.0000,-0.0419,0.9991,0.0000],[-1,0,-1,0],[9E+09,0.0000,-130.2002,9E+09,9E+09,9E+09]];
	CONST robtarget p197:=[[0.0000,-131.1231,3.7641],[0.0000,-0.0343,0.9994,0.0000],[-1,0,-1,0],[9E+09,0.0000,-131.0698,9E+09,9E+09,9E+09]];
	CONST robtarget p198:=[[0.0000,-131.0014,3.7832],[0.0000,-0.0267,0.9996,0.0000],[-1,0,-1,0],[9E+09,0.0000,-131.9413,9E+09,9E+09,9E+09]];
	CONST robtarget p199:=[[0.0000,-130.9100,3.8023],[0.0000,-0.0191,0.9998,0.0000],[-1,0,-1,0],[9E+09,0.0000,-132.8142,9E+09,9E+09,9E+09]];
	CONST robtarget p200:=[[0.0000,-130.8491,3.8214],[0.0000,-0.0114,0.9999,0.0000],[-1,0,-1,0],[9E+09,0.0000,-133.6881,9E+09,9E+09,9E+09]];
	CONST robtarget p201:=[[0.0000,-130.8186,3.8405],[0.0000,-0.0038,1.0000,0.0000],[-1,0,-1,0],[9E+09,0.0000,-134.5626,9E+09,9E+09,9E+09]];
	CONST robtarget p202:=[[0.0000,-130.8186,3.8595],[0.0000,-0.0038,-1.0000,0.0000],[-1,0,-1,0],[9E+09,0.0000,-135.4374,9E+09,9E+09,9E+09]];
	CONST robtarget p203:=[[0.0000,-130.8491,3.8786],[0.0000,-0.0114,-0.9999,0.0000],[-1,0,-1,0],[9E+09,0.0000,-136.3119,9E+09,9E+09,9E+09]];
	CONST robtarget p204:=[[0.0000,-130.9100,3.8977],[0.0000,-0.0191,-0.9998,0.0000],[-1,0,-1,0],[9E+09,0.0000,-137.1858,9E+09,9E+09,9E+09]];
	CONST robtarget p205:=[[0.0000,-131.0014,3.9168],[0.0000,-0.0267,-0.9996,0.0000],[-1,0,-1,0],[9E+09,0.0000,-138.0587,9E+09,9E+09,9E+09]];
	CONST robtarget p206:=[[0.0000,-131.1231,3.9359],[0.0000,-0.0343,-0.9994,0.0000],[-1,0,-1,0],[9E+09,0.0000,-138.9302,9E+09,9E+09,9E+09]];
	CONST robtarget p207:=[[0.0000,-131.2751,3.9550],[0.0000,-0.0419,-0.9991,0.0000],[-1,0,-1,0],[9E+09,0.0000,-139.7998,9E+09,9E+09,9E+09]];
	CONST robtarget p208:=[[0.0000,-131.4573,3.9740],[0.0000,-0.0494,-0.9988,0.0000],[-1,0,-1,0],[9E+09,0.0000,-140.6673,9E+09,9E+09,9E+09]];
	CONST robtarget p209:=[[0.0000,-131.6695,3.9931],[0.0000,-0.0570,-0.9984,0.0000],[-1,0,-1,0],[9E+09,0.0000,-141.5321,9E+09,9E+09,9E+09]];
	CONST robtarget p210:=[[0.0000,-131.9116,4.0122],[0.0000,-0.0645,-0.9979,0.0000],[-1,0,-1,0],[9E+09,0.0000,-142.3940,9E+09,9E+09,9E+09]];
	CONST robtarget p211:=[[0.0000,-132.1835,4.0313],[0.0000,-0.0720,-0.9974,0.0000],[-1,0,-1,0],[9E+09,0.0000,-143.2525,9E+09,9E+09,9E+09]];
	CONST robtarget p212:=[[0.0000,-132.4849,4.0504],[0.0000,-0.0794,-0.9968,0.0000],[-1,0,-1,0],[9E+09,0.0000,-144.1073,9E+09,9E+09,9E+09]];
	CONST robtarget p213:=[[0.0000,-132.8157,4.0695],[0.0000,-0.0868,-0.9962,0.0000],[-1,0,-1,0],[9E+09,0.0000,-144.9581,9E+09,9E+09,9E+09]];
	CONST robtarget p214:=[[0.0000,-133.1756,4.0885],[0.0000,-0.0941,-0.9956,0.0000],[-1,0,-1,0],[9E+09,0.0000,-145.8044,9E+09,9E+09,9E+09]];
	CONST robtarget p215:=[[0.0000,-133.5644,4.1076],[0.0000,-0.1015,-0.9948,0.0000],[-1,0,-1,0],[9E+09,0.0000,-146.6460,9E+09,9E+09,9E+09]];
	CONST robtarget p216:=[[0.0000,-133.9818,4.1267],[0.0000,-0.1087,-0.9941,0.0000],[-1,0,-1,0],[9E+09,0.0000,-147.4825,9E+09,9E+09,9E+09]];
	CONST robtarget p217:=[[0.0000,-134.4276,4.1458],[0.0000,-0.1159,-0.9933,0.0000],[-1,0,-1,0],[9E+09,0.0000,-148.3136,9E+09,9E+09,9E+09]];
	CONST robtarget p218:=[[0.0000,-134.9015,4.1649],[0.0000,-0.1231,-0.9924,0.0000],[-1,0,-1,0],[9E+09,0.0000,-149.1391,9E+09,9E+09,9E+09]];
	CONST robtarget p219:=[[0.0000,-135.4032,4.1840],[0.0000,-0.1302,-0.9915,0.0000],[-1,0,-1,0],[9E+09,0.0000,-149.9586,9E+09,9E+09,9E+09]];
	CONST robtarget p220:=[[0.0000,-135.9325,4.2031],[0.0000,-0.1372,-0.9905,0.0000],[-1,0,-1,0],[9E+09,0.0000,-150.7719,9E+09,9E+09,9E+09]];
	CONST robtarget p221:=[[0.0000,-136.4888,4.2221],[0.0000,-0.1442,-0.9896,0.0000],[-1,0,-1,0],[9E+09,0.0000,-151.5788,9E+09,9E+09,9E+09]];
	CONST robtarget p222:=[[0.0000,-137.0721,4.2412],[0.0000,-0.1511,-0.9885,0.0000],[-1,0,-1,0],[9E+09,0.0000,-152.3789,9E+09,9E+09,9E+09]];
	CONST robtarget p223:=[[0.0000,-137.6818,4.2603],[0.0000,-0.1579,-0.9875,0.0000],[-1,0,-1,0],[9E+09,0.0000,-153.1721,9E+09,9E+09,9E+09]];
	CONST robtarget p224:=[[0.0000,-138.3177,4.2794],[0.0000,-0.1647,-0.9863,0.0000],[-1,0,-1,0],[9E+09,0.0000,-153.9582,9E+09,9E+09,9E+09]];
	CONST robtarget p225:=[[0.0000,-138.9793,4.2985],[0.0000,-0.1714,-0.9852,0.0000],[-1,0,-1,0],[9E+09,0.0000,-154.7369,9E+09,9E+09,9E+09]];
	CONST robtarget p226:=[[0.0000,-139.6664,4.3176],[0.0000,-0.1780,-0.9840,0.0000],[-1,0,-1,0],[9E+09,0.0000,-155.5081,9E+09,9E+09,9E+09]];
	CONST robtarget p227:=[[0.0000,-140.3786,4.3366],[0.0000,-0.1846,-0.9828,0.0000],[-1,0,-1,0],[9E+09,0.0000,-156.2716,9E+09,9E+09,9E+09]];
	CONST robtarget p228:=[[0.0000,-141.1154,4.3557],[0.0000,-0.1910,-0.9816,0.0000],[-1,0,-1,0],[9E+09,0.0000,-157.0273,9E+09,9E+09,9E+09]];
	CONST robtarget p229:=[[0.0000,-141.8765,4.3748],[0.0000,-0.1974,-0.9803,0.0000],[-1,0,-1,0],[9E+09,0.0000,-157.7750,9E+09,9E+09,9E+09]];
	CONST robtarget p230:=[[0.0000,-142.6615,4.3939],[0.0000,-0.2038,-0.9790,0.0000],[-1,0,-1,0],[9E+09,0.0000,-158.5146,9E+09,9E+09,9E+09]];
	CONST robtarget p231:=[[0.0000,-143.4701,4.4130],[0.0000,-0.2100,-0.9777,0.0000],[-1,0,-1,0],[9E+09,0.0000,-159.2459,9E+09,9E+09,9E+09]];
	CONST robtarget p232:=[[0.0000,-144.3017,4.4321],[0.0000,-0.2162,-0.9764,0.0000],[-1,0,-1,0],[9E+09,0.0000,-159.9690,9E+09,9E+09,9E+09]];
	CONST robtarget p233:=[[0.0000,-145.1561,4.4511],[0.0000,-0.2223,-0.9750,0.0000],[-1,0,-1,0],[9E+09,0.0000,-160.6836,9E+09,9E+09,9E+09]];
	CONST robtarget p234:=[[0.0000,-146.0327,4.4702],[0.0000,-0.2283,-0.9736,0.0000],[-1,0,-1,0],[9E+09,0.0000,-161.3898,9E+09,9E+09,9E+09]];
	CONST robtarget p235:=[[0.0000,-146.9313,4.4893],[0.0000,-0.2342,-0.9722,0.0000],[-1,0,-1,0],[9E+09,0.0000,-162.0875,9E+09,9E+09,9E+09]];
	CONST robtarget p236:=[[0.0000,-147.8514,4.5084],[0.0000,-0.2400,-0.9708,0.0000],[-1,0,-1,0],[9E+09,0.0000,-162.7766,9E+09,9E+09,9E+09]];
	CONST robtarget p237:=[[0.0000,-148.7927,4.5275],[0.0000,-0.2458,-0.9693,0.0000],[-1,0,-1,0],[9E+09,0.0000,-163.4570,9E+09,9E+09,9E+09]];
	CONST robtarget p238:=[[0.0000,-149.7546,4.5466],[0.0000,-0.2515,-0.9679,0.0000],[-1,0,-1,0],[9E+09,0.0000,-164.1288,9E+09,9E+09,9E+09]];
	CONST robtarget p239:=[[0.0000,-150.7369,4.5656],[0.0000,-0.2571,-0.9664,0.0000],[-1,0,-1,0],[9E+09,0.0000,-164.7920,9E+09,9E+09,9E+09]];
	CONST robtarget p240:=[[0.0000,-151.7391,4.5847],[0.0000,-0.2626,-0.9649,0.0000],[-1,0,-1,0],[9E+09,0.0000,-165.4464,9E+09,9E+09,9E+09]];
	CONST robtarget p241:=[[0.0000,-152.7608,4.6038],[0.0000,-0.2680,-0.9634,0.0000],[-1,0,-1,0],[9E+09,0.0000,-166.0922,9E+09,9E+09,9E+09]];
	CONST robtarget p242:=[[0.0000,-153.8017,4.6229],[0.0000,-0.2734,-0.9619,0.0000],[-1,0,-1,0],[9E+09,0.0000,-166.7294,9E+09,9E+09,9E+09]];
	CONST robtarget p243:=[[0.0000,-154.8613,4.6420],[0.0000,-0.2786,-0.9604,0.0000],[-1,0,-1,0],[9E+09,0.0000,-167.3578,9E+09,9E+09,9E+09]];
	CONST robtarget p244:=[[0.0000,-155.9394,4.6611],[0.0000,-0.2838,-0.9589,0.0000],[-1,0,-1,0],[9E+09,0.0000,-167.9777,9E+09,9E+09,9E+09]];
	CONST robtarget p245:=[[0.0000,-157.0354,4.6802],[0.0000,-0.2889,-0.9573,0.0000],[-1,0,-1,0],[9E+09,0.0000,-168.5890,9E+09,9E+09,9E+09]];
	CONST robtarget p246:=[[0.0000,-158.1490,4.6992],[0.0000,-0.2940,-0.9558,0.0000],[-1,0,-1,0],[9E+09,0.0000,-169.1918,9E+09,9E+09,9E+09]];
	CONST robtarget p247:=[[0.0000,-159.2799,4.7183],[0.0000,-0.2989,-0.9543,0.0000],[-1,0,-1,0],[9E+09,0.0000,-169.7860,9E+09,9E+09,9E+09]];
	CONST robtarget p248:=[[0.0000,-160.4277,4.7374],[0.0000,-0.3038,-0.9527,0.0000],[-1,0,-1,0],[9E+09,0.0000,-170.3718,9E+09,9E+09,9E+09]];
	CONST robtarget p249:=[[0.0000,-161.5921,4.7565],[0.0000,-0.3086,-0.9512,0.0000],[-1,0,-1,0],[9E+09,0.0000,-170.9493,9E+09,9E+09,9E+09]];
	CONST robtarget p250:=[[0.0000,-162.7726,4.7756],[0.0000,-0.3133,-0.9496,0.0000],[-1,0,-1,0],[9E+09,0.0000,-171.5184,9E+09,9E+09,9E+09]];
	CONST robtarget p251:=[[0.0000,-163.9689,4.7947],[0.0000,-0.3180,-0.9481,0.0000],[-1,0,-1,0],[9E+09,0.0000,-172.0793,9E+09,9E+09,9E+09]];
	CONST robtarget p252:=[[0.0000,-165.1807,4.8137],[0.0000,-0.3225,-0.9466,0.0000],[-1,0,-1,0],[9E+09,0.0000,-172.6319,9E+09,9E+09,9E+09]];
	CONST robtarget p253:=[[0.0000,-166.4077,4.8328],[0.0000,-0.3270,-0.9450,0.0000],[-1,0,-1,0],[9E+09,0.0000,-173.1765,9E+09,9E+09,9E+09]];
	CONST robtarget p254:=[[0.0000,-167.6495,4.8519],[0.0000,-0.3314,-0.9435,0.0000],[-1,0,-1,0],[9E+09,0.0000,-173.7131,9E+09,9E+09,9E+09]];
	CONST robtarget p255:=[[0.0000,-168.9057,4.8710],[0.0000,-0.3358,-0.9419,0.0000],[-1,0,-1,0],[9E+09,0.0000,-174.2417,9E+09,9E+09,9E+09]];
	CONST robtarget p256:=[[0.0000,-170.1762,4.8901],[0.0000,-0.3401,-0.9404,0.0000],[-1,0,-1,0],[9E+09,0.0000,-174.7625,9E+09,9E+09,9E+09]];
	CONST robtarget p257:=[[0.0000,-171.4604,4.9092],[0.0000,-0.3443,-0.9389,0.0000],[-1,0,-1,0],[9E+09,0.0000,-175.2755,9E+09,9E+09,9E+09]];
	CONST robtarget p258:=[[0.0000,-172.7582,4.9282],[0.0000,-0.3484,-0.9373,0.0000],[-1,0,-1,0],[9E+09,0.0000,-175.7809,9E+09,9E+09,9E+09]];
	CONST robtarget p259:=[[0.0000,-174.0693,4.9473],[0.0000,-0.3525,-0.9358,0.0000],[-1,0,-1,0],[9E+09,0.0000,-176.2787,9E+09,9E+09,9E+09]];
	CONST robtarget p260:=[[0.0000,-175.3933,4.9664],[0.0000,-0.3565,-0.9343,0.0000],[-1,0,-1,0],[9E+09,0.0000,-176.7690,9E+09,9E+09,9E+09]];
	CONST robtarget p261:=[[0.0000,-176.7300,4.9855],[0.0000,-0.3604,-0.9328,0.0000],[-1,0,-1,0],[9E+09,0.0000,-177.2519,9E+09,9E+09,9E+09]];
	CONST robtarget p262:=[[0.0000,-178.0790,5.0046],[0.0000,-0.3643,-0.9313,0.0000],[-1,0,-1,0],[9E+09,0.0000,-177.7276,9E+09,9E+09,9E+09]];
	CONST robtarget p263:=[[0.0000,-179.4401,5.0237],[0.0000,-0.3681,-0.9298,0.0000],[-1,0,-1,0],[9E+09,0.0000,-178.1960,9E+09,9E+09,9E+09]];
	CONST robtarget p264:=[[0.0000,-180.8130,5.0427],[0.0000,-0.3718,-0.9283,0.0000],[-1,0,-1,0],[9E+09,0.0000,-178.6574,9E+09,9E+09,9E+09]];
	CONST robtarget p265:=[[0.0000,-182.1975,5.0618],[0.0000,-0.3755,-0.9268,0.0000],[-1,0,-1,0],[9E+09,0.0000,-179.1118,9E+09,9E+09,9E+09]];
	CONST robtarget p266:=[[0.0000,-183.5932,5.0809],[0.0000,-0.3791,-0.9253,0.0000],[-1,0,-1,0],[9E+09,0.0000,-179.5593,9E+09,9E+09,9E+09]];
	CONST robtarget p267:=[[0.0000,-185.0000,5.1000],[0.0000,-0.3827,0.9239,0.0000],[-1,0,-1,0],[9E+09,0.0000,-180.0000,9E+09,9E+09,9E+09]];
	CONST robtarget p268:=[[0.0000,-183.5932,5.1191],[0.0000,-0.3791,0.9253,0.0000],[-1,0,-1,0],[9E+09,0.0000,-180.4407,9E+09,9E+09,9E+09]];
	CONST robtarget p269:=[[0.0000,-182.1975,5.1382],[0.0000,-0.3755,0.9268,0.0000],[-1,0,-1,0],[9E+09,0.0000,-180.8882,9E+09,9E+09,9E+09]];
	CONST robtarget p270:=[[0.0000,-180.8130,5.1573],[0.0000,-0.3718,0.9283,0.0000],[-1,0,-1,0],[9E+09,0.0000,-181.3426,9E+09,9E+09,9E+09]];
	CONST robtarget p271:=[[0.0000,-179.4401,5.1763],[0.0000,-0.3681,0.9298,0.0000],[-1,0,-1,0],[9E+09,0.0000,-181.8040,9E+09,9E+09,9E+09]];
	CONST robtarget p272:=[[0.0000,-178.0790,5.1954],[0.0000,-0.3643,0.9313,0.0000],[-1,0,-1,0],[9E+09,0.0000,-182.2724,9E+09,9E+09,9E+09]];
	CONST robtarget p273:=[[0.0000,-176.7300,5.2145],[0.0000,-0.3604,0.9328,0.0000],[-1,0,-1,0],[9E+09,0.0000,-182.7481,9E+09,9E+09,9E+09]];
	CONST robtarget p274:=[[0.0000,-175.3933,5.2336],[0.0000,-0.3565,0.9343,0.0000],[-1,0,-1,0],[9E+09,0.0000,-183.2310,9E+09,9E+09,9E+09]];
	CONST robtarget p275:=[[0.0000,-174.0693,5.2527],[0.0000,-0.3525,0.9358,0.0000],[-1,0,-1,0],[9E+09,0.0000,-183.7213,9E+09,9E+09,9E+09]];
	CONST robtarget p276:=[[0.0000,-172.7582,5.2718],[0.0000,-0.3484,0.9373,0.0000],[-1,0,-1,0],[9E+09,0.0000,-184.2191,9E+09,9E+09,9E+09]];
	CONST robtarget p277:=[[0.0000,-171.4604,5.2908],[0.0000,-0.3443,0.9389,0.0000],[-1,0,-1,0],[9E+09,0.0000,-184.7245,9E+09,9E+09,9E+09]];
	CONST robtarget p278:=[[0.0000,-170.1762,5.3099],[0.0000,-0.3401,0.9404,0.0000],[-1,0,-1,0],[9E+09,0.0000,-185.2375,9E+09,9E+09,9E+09]];
	CONST robtarget p279:=[[0.0000,-168.9057,5.3290],[0.0000,-0.3358,0.9419,0.0000],[-1,0,-1,0],[9E+09,0.0000,-185.7583,9E+09,9E+09,9E+09]];
	CONST robtarget p280:=[[0.0000,-167.6495,5.3481],[0.0000,-0.3314,0.9435,0.0000],[-1,0,-1,0],[9E+09,0.0000,-186.2869,9E+09,9E+09,9E+09]];
	CONST robtarget p281:=[[0.0000,-166.4077,5.3672],[0.0000,-0.3270,0.9450,0.0000],[-1,0,-1,0],[9E+09,0.0000,-186.8235,9E+09,9E+09,9E+09]];
	CONST robtarget p282:=[[0.0000,-165.1807,5.3863],[0.0000,-0.3225,0.9466,0.0000],[-1,0,-1,0],[9E+09,0.0000,-187.3681,9E+09,9E+09,9E+09]];
	CONST robtarget p283:=[[0.0000,-163.9689,5.4053],[0.0000,-0.3180,0.9481,0.0000],[-1,0,-1,0],[9E+09,0.0000,-187.9207,9E+09,9E+09,9E+09]];
	CONST robtarget p284:=[[0.0000,-162.7726,5.4244],[0.0000,-0.3133,0.9496,0.0000],[-1,0,-1,0],[9E+09,0.0000,-188.4816,9E+09,9E+09,9E+09]];
	CONST robtarget p285:=[[0.0000,-161.5921,5.4435],[0.0000,-0.3086,0.9512,0.0000],[-1,0,-1,0],[9E+09,0.0000,-189.0507,9E+09,9E+09,9E+09]];
	CONST robtarget p286:=[[0.0000,-160.4277,5.4626],[0.0000,-0.3038,0.9527,0.0000],[-1,0,-1,0],[9E+09,0.0000,-189.6282,9E+09,9E+09,9E+09]];
	CONST robtarget p287:=[[0.0000,-159.2799,5.4817],[0.0000,-0.2989,0.9543,0.0000],[-1,0,-1,0],[9E+09,0.0000,-190.2140,9E+09,9E+09,9E+09]];
	CONST robtarget p288:=[[0.0000,-158.1490,5.5008],[0.0000,-0.2940,0.9558,0.0000],[-1,0,-1,0],[9E+09,0.0000,-190.8082,9E+09,9E+09,9E+09]];
	CONST robtarget p289:=[[0.0000,-157.0354,5.5198],[0.0000,-0.2889,0.9573,0.0000],[-1,0,-1,0],[9E+09,0.0000,-191.4110,9E+09,9E+09,9E+09]];
	CONST robtarget p290:=[[0.0000,-155.9394,5.5389],[0.0000,-0.2838,0.9589,0.0000],[-1,0,-1,0],[9E+09,0.0000,-192.0223,9E+09,9E+09,9E+09]];
	CONST robtarget p291:=[[0.0000,-154.8613,5.5580],[0.0000,-0.2786,0.9604,0.0000],[-1,0,-1,0],[9E+09,0.0000,-192.6422,9E+09,9E+09,9E+09]];
	CONST robtarget p292:=[[0.0000,-153.8017,5.5771],[0.0000,-0.2734,0.9619,0.0000],[-1,0,-1,0],[9E+09,0.0000,-193.2706,9E+09,9E+09,9E+09]];
	CONST robtarget p293:=[[0.0000,-152.7608,5.5962],[0.0000,-0.2680,0.9634,0.0000],[-1,0,-1,0],[9E+09,0.0000,-193.9078,9E+09,9E+09,9E+09]];
	CONST robtarget p294:=[[0.0000,-151.7391,5.6153],[0.0000,-0.2626,0.9649,0.0000],[-1,0,-1,0],[9E+09,0.0000,-194.5536,9E+09,9E+09,9E+09]];
	CONST robtarget p295:=[[0.0000,-150.7369,5.6344],[0.0000,-0.2571,0.9664,0.0000],[-1,0,-1,0],[9E+09,0.0000,-195.2080,9E+09,9E+09,9E+09]];
	CONST robtarget p296:=[[0.0000,-149.7546,5.6534],[0.0000,-0.2515,0.9679,0.0000],[-1,0,-1,0],[9E+09,0.0000,-195.8712,9E+09,9E+09,9E+09]];
	CONST robtarget p297:=[[0.0000,-148.7927,5.6725],[0.0000,-0.2458,0.9693,0.0000],[-1,0,-1,0],[9E+09,0.0000,-196.5430,9E+09,9E+09,9E+09]];
	CONST robtarget p298:=[[0.0000,-147.8514,5.6916],[0.0000,-0.2400,0.9708,0.0000],[-1,0,-1,0],[9E+09,0.0000,-197.2234,9E+09,9E+09,9E+09]];
	CONST robtarget p299:=[[0.0000,-146.9313,5.7107],[0.0000,-0.2342,0.9722,0.0000],[-1,0,-1,0],[9E+09,0.0000,-197.9125,9E+09,9E+09,9E+09]];
	CONST robtarget p300:=[[0.0000,-146.0327,5.7298],[0.0000,-0.2283,0.9736,0.0000],[-1,0,-1,0],[9E+09,0.0000,-198.6102,9E+09,9E+09,9E+09]];
	CONST robtarget p301:=[[0.0000,-145.1561,5.7489],[0.0000,-0.2223,0.9750,0.0000],[-1,0,-1,0],[9E+09,0.0000,-199.3164,9E+09,9E+09,9E+09]];
	CONST robtarget p302:=[[0.0000,-144.3017,5.7679],[0.0000,-0.2162,0.9764,0.0000],[-1,0,-1,0],[9E+09,0.0000,-200.0310,9E+09,9E+09,9E+09]];
	CONST robtarget p303:=[[0.0000,-143.4701,5.7870],[0.0000,-0.2100,0.9777,0.0000],[-1,0,-1,0],[9E+09,0.0000,-200.7541,9E+09,9E+09,9E+09]];
	CONST robtarget p304:=[[0.0000,-142.6615,5.8061],[0.0000,-0.2038,0.9790,0.0000],[-1,0,-1,0],[9E+09,0.0000,-201.4854,9E+09,9E+09,9E+09]];
	CONST robtarget p305:=[[0.0000,-141.8765,5.8252],[0.0000,-0.1974,0.9803,0.0000],[-1,0,-1,0],[9E+09,0.0000,-202.2250,9E+09,9E+09,9E+09]];
	CONST robtarget p306:=[[0.0000,-141.1154,5.8443],[0.0000,-0.1910,0.9816,0.0000],[-1,0,-1,0],[9E+09,0.0000,-202.9727,9E+09,9E+09,9E+09]];
	CONST robtarget p307:=[[0.0000,-140.3786,5.8634],[0.0000,-0.1846,0.9828,0.0000],[-1,0,-1,0],[9E+09,0.0000,-203.7284,9E+09,9E+09,9E+09]];
	CONST robtarget p308:=[[0.0000,-139.6664,5.8824],[0.0000,-0.1780,0.9840,0.0000],[-1,0,-1,0],[9E+09,0.0000,-204.4919,9E+09,9E+09,9E+09]];
	CONST robtarget p309:=[[0.0000,-138.9793,5.9015],[0.0000,-0.1714,0.9852,0.0000],[-1,0,-1,0],[9E+09,0.0000,-205.2631,9E+09,9E+09,9E+09]];
	CONST robtarget p310:=[[0.0000,-138.3177,5.9206],[0.0000,-0.1647,0.9863,0.0000],[-1,0,-1,0],[9E+09,0.0000,-206.0418,9E+09,9E+09,9E+09]];
	CONST robtarget p311:=[[0.0000,-137.6818,5.9397],[0.0000,-0.1579,0.9875,0.0000],[-1,0,-1,0],[9E+09,0.0000,-206.8279,9E+09,9E+09,9E+09]];
	CONST robtarget p312:=[[0.0000,-137.0721,5.9588],[0.0000,-0.1511,0.9885,0.0000],[-1,0,-1,0],[9E+09,0.0000,-207.6211,9E+09,9E+09,9E+09]];
	CONST robtarget p313:=[[0.0000,-136.4888,5.9779],[0.0000,-0.1442,0.9896,0.0000],[-1,0,-1,0],[9E+09,0.0000,-208.4212,9E+09,9E+09,9E+09]];
	CONST robtarget p314:=[[0.0000,-135.9325,5.9969],[0.0000,-0.1372,0.9905,0.0000],[-1,0,-1,0],[9E+09,0.0000,-209.2281,9E+09,9E+09,9E+09]];
	CONST robtarget p315:=[[0.0000,-135.4032,6.0160],[0.0000,-0.1302,0.9915,0.0000],[-1,0,-1,0],[9E+09,0.0000,-210.0414,9E+09,9E+09,9E+09]];
	CONST robtarget p316:=[[0.0000,-134.9015,6.0351],[0.0000,-0.1231,0.9924,0.0000],[-1,0,-1,0],[9E+09,0.0000,-210.8609,9E+09,9E+09,9E+09]];
	CONST robtarget p317:=[[0.0000,-134.4276,6.0542],[0.0000,-0.1159,0.9933,0.0000],[-1,0,-1,0],[9E+09,0.0000,-211.6864,9E+09,9E+09,9E+09]];
	CONST robtarget p318:=[[0.0000,-133.9818,6.0733],[0.0000,-0.1087,0.9941,0.0000],[-1,0,-1,0],[9E+09,0.0000,-212.5175,9E+09,9E+09,9E+09]];
	CONST robtarget p319:=[[0.0000,-133.5644,6.0924],[0.0000,-0.1015,0.9948,0.0000],[-1,0,-1,0],[9E+09,0.0000,-213.3540,9E+09,9E+09,9E+09]];
	CONST robtarget p320:=[[0.0000,-133.1756,6.1115],[0.0000,-0.0941,0.9956,0.0000],[-1,0,-1,0],[9E+09,0.0000,-214.1956,9E+09,9E+09,9E+09]];
	CONST robtarget p321:=[[0.0000,-132.8157,6.1305],[0.0000,-0.0868,0.9962,0.0000],[-1,0,-1,0],[9E+09,0.0000,-215.0419,9E+09,9E+09,9E+09]];
	CONST robtarget p322:=[[0.0000,-132.4849,6.1496],[0.0000,-0.0794,0.9968,0.0000],[-1,0,-1,0],[9E+09,0.0000,-215.8927,9E+09,9E+09,9E+09]];
	CONST robtarget p323:=[[0.0000,-132.1835,6.1687],[0.0000,-0.0720,0.9974,0.0000],[-1,0,-1,0],[9E+09,0.0000,-216.7475,9E+09,9E+09,9E+09]];
	CONST robtarget p324:=[[0.0000,-131.9116,6.1878],[0.0000,-0.0645,0.9979,0.0000],[-1,0,-1,0],[9E+09,0.0000,-217.6060,9E+09,9E+09,9E+09]];
	CONST robtarget p325:=[[0.0000,-131.6695,6.2069],[0.0000,-0.0570,0.9984,0.0000],[-1,0,-1,0],[9E+09,0.0000,-218.4679,9E+09,9E+09,9E+09]];
	CONST robtarget p326:=[[0.0000,-131.4573,6.2260],[0.0000,-0.0494,0.9988,0.0000],[-1,0,-1,0],[9E+09,0.0000,-219.3327,9E+09,9E+09,9E+09]];
	CONST robtarget p327:=[[0.0000,-131.2751,6.2450],[0.0000,-0.0419,0.9991,0.0000],[-1,0,-1,0],[9E+09,0.0000,-220.2002,9E+09,9E+09,9E+09]];
	CONST robtarget p328:=[[0.0000,-131.1231,6.2641],[0.0000,-0.0343,0.9994,0.0000],[-1,0,-1,0],[9E+09,0.0000,-221.0698,9E+09,9E+09,9E+09]];
	CONST robtarget p329:=[[0.0000,-131.0014,6.2832],[0.0000,-0.0267,0.9996,0.0000],[-1,0,-1,0],[9E+09,0.0000,-221.9413,9E+09,9E+09,9E+09]];
	CONST robtarget p330:=[[0.0000,-130.9100,6.3023],[0.0000,-0.0191,0.9998,0.0000],[-1,0,-1,0],[9E+09,0.0000,-222.8142,9E+09,9E+09,9E+09]];
	CONST robtarget p331:=[[0.0000,-130.8491,6.3214],[0.0000,-0.0114,0.9999,0.0000],[-1,0,-1,0],[9E+09,0.0000,-223.6881,9E+09,9E+09,9E+09]];
	CONST robtarget p332:=[[0.0000,-130.8186,6.3405],[0.0000,-0.0038,1.0000,0.0000],[-1,0,-1,0],[9E+09,0.0000,-224.5626,9E+09,9E+09,9E+09]];
	CONST robtarget p333:=[[0.0000,-130.8186,6.3595],[0.0000,-0.0038,-1.0000,0.0000],[-1,0,-1,0],[9E+09,0.0000,-225.4374,9E+09,9E+09,9E+09]];
	CONST robtarget p334:=[[0.0000,-130.8491,6.3786],[0.0000,-0.0114,-0.9999,0.0000],[-1,0,-1,0],[9E+09,0.0000,-226.3119,9E+09,9E+09,9E+09]];
	CONST robtarget p335:=[[0.0000,-130.9100,6.3977],[0.0000,-0.0191,-0.9998,0.0000],[-1,0,-1,0],[9E+09,0.0000,-227.1858,9E+09,9E+09,9E+09]];
	CONST robtarget p336:=[[0.0000,-131.0014,6.4168],[0.0000,-0.0267,-0.9996,0.0000],[-1,0,-1,0],[9E+09,0.0000,-228.0587,9E+09,9E+09,9E+09]];
	CONST robtarget p337:=[[0.0000,-131.1231,6.4359],[0.0000,-0.0343,-0.9994,0.0000],[-1,0,-1,0],[9E+09,0.0000,-228.9302,9E+09,9E+09,9E+09]];
	CONST robtarget p338:=[[0.0000,-131.2751,6.4550],[0.0000,-0.0419,-0.9991,0.0000],[-1,0,-1,0],[9E+09,0.0000,-229.7998,9E+09,9E+09,9E+09]];
	CONST robtarget p339:=[[0.0000,-131.4573,6.4740],[0.0000,-0.0494,-0.9988,0.0000],[-1,0,-1,0],[9E+09,0.0000,-230.6673,9E+09,9E+09,9E+09]];
	CONST robtarget p340:=[[0.0000,-131.6695,6.4931],[0.0000,-0.0570,-0.9984,0.0000],[-1,0,-1,0],[9E+09,0.0000,-231.5321,9E+09,9E+09,9E+09]];
	CONST robtarget p341:=[[0.0000,-131.9116,6.5122],[0.0000,-0.0645,-0.9979,0.0000],[-1,0,-1,0],[9E+09,0.0000,-232.3940,9E+09,9E+09,9E+09]];
	CONST robtarget p342:=[[0.0000,-132.1835,6.5313],[0.0000,-0.0720,-0.9974,0.0000],[-1,0,-1,0],[9E+09,0.0000,-233.2525,9E+09,9E+09,9E+09]];
	CONST robtarget p343:=[[0.0000,-132.4849,6.5504],[0.0000,-0.0794,-0.9968,0.0000],[-1,0,-1,0],[9E+09,0.0000,-234.1073,9E+09,9E+09,9E+09]];
	CONST robtarget p344:=[[0.0000,-132.8157,6.5695],[0.0000,-0.0868,-0.9962,0.0000],[-1,0,-1,0],[9E+09,0.0000,-234.9581,9E+09,9E+09,9E+09]];
	CONST robtarget p345:=[[0.0000,-133.1756,6.5885],[0.0000,-0.0941,-0.9956,0.0000],[-1,0,-1,0],[9E+09,0.0000,-235.8044,9E+09,9E+09,9E+09]];
	CONST robtarget p346:=[[0.0000,-133.5644,6.6076],[0.0000,-0.1015,-0.9948,0.0000],[-1,0,-1,0],[9E+09,0.0000,-236.6460,9E+09,9E+09,9E+09]];
	CONST robtarget p347:=[[0.0000,-133.9818,6.6267],[0.0000,-0.1087,-0.9941,0.0000],[-1,0,-1,0],[9E+09,0.0000,-237.4825,9E+09,9E+09,9E+09]];
	CONST robtarget p348:=[[0.0000,-134.4276,6.6458],[0.0000,-0.1159,-0.9933,0.0000],[-1,0,-1,0],[9E+09,0.0000,-238.3136,9E+09,9E+09,9E+09]];
	CONST robtarget p349:=[[0.0000,-134.9015,6.6649],[0.0000,-0.1231,-0.9924,0.0000],[-1,0,-1,0],[9E+09,0.0000,-239.1391,9E+09,9E+09,9E+09]];
	CONST robtarget p350:=[[0.0000,-135.4032,6.6840],[0.0000,-0.1302,-0.9915,0.0000],[-1,0,-1,0],[9E+09,0.0000,-239.9586,9E+09,9E+09,9E+09]];
	CONST robtarget p351:=[[0.0000,-135.9325,6.7031],[0.0000,-0.1372,-0.9905,0.0000],[-1,0,-1,0],[9E+09,0.0000,-240.7719,9E+09,9E+09,9E+09]];
	CONST robtarget p352:=[[0.0000,-136.4888,6.7221],[0.0000,-0.1442,-0.9896,0.0000],[-1,0,-1,0],[9E+09,0.0000,-241.5788,9E+09,9E+09,9E+09]];
	CONST robtarget p353:=[[0.0000,-137.0721,6.7412],[0.0000,-0.1511,-0.9885,0.0000],[-1,0,-1,0],[9E+09,0.0000,-242.3789,9E+09,9E+09,9E+09]];
	CONST robtarget p354:=[[0.0000,-137.6818,6.7603],[0.0000,-0.1579,-0.9875,0.0000],[-1,0,-1,0],[9E+09,0.0000,-243.1721,9E+09,9E+09,9E+09]];
	CONST robtarget p355:=[[0.0000,-138.3177,6.7794],[0.0000,-0.1647,-0.9863,0.0000],[-1,0,-1,0],[9E+09,0.0000,-243.9582,9E+09,9E+09,9E+09]];
	CONST robtarget p356:=[[0.0000,-138.9793,6.7985],[0.0000,-0.1714,-0.9852,0.0000],[-1,0,-1,0],[9E+09,0.0000,-244.7369,9E+09,9E+09,9E+09]];
	CONST robtarget p357:=[[0.0000,-139.6664,6.8176],[0.0000,-0.1780,-0.9840,0.0000],[-1,0,-1,0],[9E+09,0.0000,-245.5081,9E+09,9E+09,9E+09]];
	CONST robtarget p358:=[[0.0000,-140.3786,6.8366],[0.0000,-0.1846,-0.9828,0.0000],[-1,0,-1,0],[9E+09,0.0000,-246.2716,9E+09,9E+09,9E+09]];
	CONST robtarget p359:=[[0.0000,-141.1154,6.8557],[0.0000,-0.1910,-0.9816,0.0000],[-1,0,-1,0],[9E+09,0.0000,-247.0273,9E+09,9E+09,9E+09]];
	CONST robtarget p360:=[[0.0000,-141.8765,6.8748],[0.0000,-0.1974,-0.9803,0.0000],[-1,0,-1,0],[9E+09,0.0000,-247.7750,9E+09,9E+09,9E+09]];
	CONST robtarget p361:=[[0.0000,-142.6615,6.8939],[0.0000,-0.2038,-0.9790,0.0000],[-1,0,-1,0],[9E+09,0.0000,-248.5146,9E+09,9E+09,9E+09]];
	CONST robtarget p362:=[[0.0000,-143.4701,6.9130],[0.0000,-0.2100,-0.9777,0.0000],[-1,0,-1,0],[9E+09,0.0000,-249.2459,9E+09,9E+09,9E+09]];
	CONST robtarget p363:=[[0.0000,-144.3017,6.9321],[0.0000,-0.2162,-0.9764,0.0000],[-1,0,-1,0],[9E+09,0.0000,-249.9690,9E+09,9E+09,9E+09]];
	CONST robtarget p364:=[[0.0000,-145.1561,6.9511],[0.0000,-0.2223,-0.9750,0.0000],[-1,0,-1,0],[9E+09,0.0000,-250.6836,9E+09,9E+09,9E+09]];
	CONST robtarget p365:=[[0.0000,-146.0327,6.9702],[0.0000,-0.2283,-0.9736,0.0000],[-1,0,-1,0],[9E+09,0.0000,-251.3898,9E+09,9E+09,9E+09]];
	CONST robtarget p366:=[[0.0000,-146.9313,6.9893],[0.0000,-0.2342,-0.9722,0.0000],[-1,0,-1,0],[9E+09,0.0000,-252.0875,9E+09,9E+09,9E+09]];
	CONST robtarget p367:=[[0.0000,-147.8514,7.0084],[0.0000,-0.2400,-0.9708,0.0000],[-1,0,-1,0],[9E+09,0.0000,-252.7766,9E+09,9E+09,9E+09]];
	CONST robtarget p368:=[[0.0000,-148.7927,7.0275],[0.0000,-0.2458,-0.9693,0.0000],[-1,0,-1,0],[9E+09,0.0000,-253.4570,9E+09,9E+09,9E+09]];
	CONST robtarget p369:=[[0.0000,-149.7546,7.0466],[0.0000,-0.2515,-0.9679,0.0000],[-1,0,-1,0],[9E+09,0.0000,-254.1288,9E+09,9E+09,9E+09]];
	CONST robtarget p370:=[[0.0000,-150.7369,7.0656],[0.0000,-0.2571,-0.9664,0.0000],[-1,0,-1,0],[9E+09,0.0000,-254.7920,9E+09,9E+09,9E+09]];
	CONST robtarget p371:=[[0.0000,-151.7391,7.0847],[0.0000,-0.2626,-0.9649,0.0000],[-1,0,-1,0],[9E+09,0.0000,-255.4464,9E+09,9E+09,9E+09]];
	CONST robtarget p372:=[[0.0000,-152.7608,7.1038],[0.0000,-0.2680,-0.9634,0.0000],[-1,0,-1,0],[9E+09,0.0000,-256.0922,9E+09,9E+09,9E+09]];
	CONST robtarget p373:=[[0.0000,-153.8017,7.1229],[0.0000,-0.2734,-0.9619,0.0000],[-1,0,-1,0],[9E+09,0.0000,-256.7294,9E+09,9E+09,9E+09]];
	CONST robtarget p374:=[[0.0000,-154.8613,7.1420],[0.0000,-0.2786,-0.9604,0.0000],[-1,0,-1,0],[9E+09,0.0000,-257.3578,9E+09,9E+09,9E+09]];
	CONST robtarget p375:=[[0.0000,-155.9394,7.1611],[0.0000,-0.2838,-0.9589,0.0000],[-1,0,-1,0],[9E+09,0.0000,-257.9777,9E+09,9E+09,9E+09]];
	CONST robtarget p376:=[[0.0000,-157.0354,7.1802],[0.0000,-0.2889,-0.9573,0.0000],[-1,0,-1,0],[9E+09,0.0000,-258.5890,9E+09,9E+09,9E+09]];
	CONST robtarget p377:=[[0.0000,-158.1490,7.1992],[0.0000,-0.2940,-0.9558,0.0000],[-1,0,-1,0],[9E+09,0.0000,-259.1918,9E+09,9E+09,9E+09]];
	CONST robtarget p378:=[[0.0000,-159.2799,7.2183],[0.0000,-0.2989,-0.9543,0.0000],[-1,0,-1,0],[9E+09,0.0000,-259.7860,9E+09,9E+09,9E+09]];
	CONST robtarget p379:=[[0.0000,-160.4277,7.2374],[0.0000,-0.3038,-0.9527,0.0000],[-1,0,-1,0],[9E+09,0.0000,-260.3718,9E+09,9E+09,9E+09]];
	CONST robtarget p380:=[[0.0000,-161.5921,7.2565],[0.0000,-0.3086,-0.9512,0.0000],[-1,0,-1,0],[9E+09,0.0000,-260.9493,9E+09,9E+09,9E+09]];
	CONST robtarget p381:=[[0.0000,-162.7726,7.2756],[0.0000,-0.3133,-0.9496,0.0000],[-1,0,-1,0],[9E+09,0.0000,-261.5184,9E+09,9E+09,9E+09]];
	CONST robtarget p382:=[[0.0000,-163.9689,7.2947],[0.0000,-0.3180,-0.9481,0.0000],[-1,0,-1,0],[9E+09,0.0000,-262.0793,9E+09,9E+09,9E+09]];
	CONST robtarget p383:=[[0.0000,-165.1807,7.3137],[0.0000,-0.3225,-0.9466,0.0000],[-1,0,-1,0],[9E+09,0.0000,-262.6319,9E+09,9E+09,9E+09]];
	CONST robtarget p384:=[[0.0000,-166.4077,7.3328],[0.0000,-0.3270,-0.9450,0.0000],[-1,0,-1,0],[9E+09,0.0000,-263.1765,9E+09,9E+09,9E+09]];
	CONST robtarget p385:=[[0.0000,-167.6495,7.3519],[0.0000,-0.3314,-0.9435,0.0000],[-1,0,-1,0],[9E+09,0.0000,-263.7131,9E+09,9E+09,9E+09]];
	CONST robtarget p386:=[[0.0000,-168.9057,7.3710],[0.0000,-0.3358,-0.9419,0.0000],[-1,0,-1,0],[9E+09,0.0000,-264.2417,9E+09,9E+09,9E+09]];
	CONST robtarget p387:=[[0.0000,-170.1762,7.3901],[0.0000,-0.3401,-0.9404,0.0000],[-1,0,-1,0],[9E+09,0.0000,-264.7625,9E+09,9E+09,9E+09]];
	CONST robtarget p388:=[[0.0000,-171.4604,7.4092],[0.0000,-0.3443,-0.9389,0.0000],[-1,0,-1,0],[9E+09,0.0000,-265.2755,9E+09,9E+09,9E+09]];
	CONST robtarget p389:=[[0.0000,-172.7582,7.4282],[0.0000,-0.3484,-0.9373,0.0000],[-1,0,-1,0],[9E+09,0.0000,-265.7809,9E+09,9E+09,9E+09]];
	CONST robtarget p390:=[[0.0000,-174.0693,7.4473],[0.0000,-0.3525,-0.9358,0.0000],[-1,0,-1,0],[9E+09,0.0000,-266.2787,9E+09,9E+09,9E+09]];
	CONST robtarget p391:=[[0.0000,-175.3933,7.4664],[0.0000,-0.3565,-0.9343,0.0000],[-1,0,-1,0],[9E+09,0.0000,-266.7690,9E+09,9E+09,9E+09]];
	CONST robtarget p392:=[[0.0000,-176.7300,7.4855],[0.0000,-0.3604,-0.9328,0.0000],[-1,0,-1,0],[9E+09,0.0000,-267.2519,9E+09,9E+09,9E+09]];
	CONST robtarget p393:=[[0.0000,-178.0790,7.5046],[0.0000,-0.3643,-0.9313,0.0000],[-1,0,-1,0],[9E+09,0.0000,-267.7276,9E+09,9E+09,9E+09]];
	CONST robtarget p394:=[[0.0000,-179.4401,7.5237],[0.0000,-0.3681,-0.9298,0.0000],[-1,0,-1,0],[9E+09,0.0000,-268.1960,9E+09,9E+09,9E+09]];
	CONST robtarget p395:=[[0.0000,-180.8130,7.5427],[0.0000,-0.3718,-0.9283,0.0000],[-1,0,-1,0],[9E+09,0.0000,-268.6574,9E+09,9E+09,9E+09]];
	CONST robtarget p396:=[[0.0000,-182.1975,7.5618],[0.0000,-0.3755,-0.9268,0.0000],[-1,0,-1,0],[9E+09,0.0000,-269.1118,9E+09,9E+09,9E+09]];
	CONST robtarget p397:=[[0.0000,-183.5932,7.5809],[0.0000,-0.3791,-0.9253,0.0000],[-1,0,-1,0],[9E+09,0.0000,-269.5593,9E+09,9E+09,9E+09]];
	CONST robtarget p398:=[[0.0000,-185.0000,7.6000],[0.0000,-0.3827,0.9239,0.0000],[-1,0,-1,0],[9E+09,0.0000,-270.0000,9E+09,9E+09,9E+09]];
	CONST robtarget p399:=[[0.0000,-183.5932,7.6191],[0.0000,-0.3791,0.9253,0.0000],[-1,0,-1,0],[9E+09,0.0000,-270.4407,9E+09,9E+09,9E+09]];
	CONST robtarget p400:=[[0.0000,-182.1975,7.6382],[0.0000,-0.3755,0.9268,0.0000],[-1,0,-1,0],[9E+09,0.0000,-270.8882,9E+09,9E+09,9E+09]];
	CONST robtarget p401:=[[0.0000,-180.8130,7.6573],[0.0000,-0.3718,0.9283,0.0000],[-1,0,-1,0],[9E+09,0.0000,-271.3426,9E+09,9E+09,9E+09]];
	CONST robtarget p402:=[[0.0000,-179.4401,7.6763],[0.0000,-0.3681,0.9298,0.0000],[-1,0,-1,0],[9E+09,0.0000,-271.8040,9E+09,9E+09,9E+09]];
	CONST robtarget p403:=[[0.0000,-178.0790,7.6954],[0.0000,-0.3643,0.9313,0.0000],[-1,0,-1,0],[9E+09,0.0000,-272.2724,9E+09,9E+09,9E+09]];
	CONST robtarget p404:=[[0.0000,-176.7300,7.7145],[0.0000,-0.3604,0.9328,0.0000],[-1,0,-1,0],[9E+09,0.0000,-272.7481,9E+09,9E+09,9E+09]];
	CONST robtarget p405:=[[0.0000,-175.3933,7.7336],[0.0000,-0.3565,0.9343,0.0000],[-1,0,-1,0],[9E+09,0.0000,-273.2310,9E+09,9E+09,9E+09]];
	CONST robtarget p406:=[[0.0000,-174.0693,7.7527],[0.0000,-0.3525,0.9358,0.0000],[-1,0,-1,0],[9E+09,0.0000,-273.7213,9E+09,9E+09,9E+09]];
	CONST robtarget p407:=[[0.0000,-172.7582,7.7718],[0.0000,-0.3484,0.9373,0.0000],[-1,0,-1,0],[9E+09,0.0000,-274.2191,9E+09,9E+09,9E+09]];
	CONST robtarget p408:=[[0.0000,-171.4604,7.7908],[0.0000,-0.3443,0.9389,0.0000],[-1,0,-1,0],[9E+09,0.0000,-274.7245,9E+09,9E+09,9E+09]];
	CONST robtarget p409:=[[0.0000,-170.1762,7.8099],[0.0000,-0.3401,0.9404,0.0000],[-1,0,-1,0],[9E+09,0.0000,-275.2375,9E+09,9E+09,9E+09]];
	CONST robtarget p410:=[[0.0000,-168.9057,7.8290],[0.0000,-0.3358,0.9419,0.0000],[-1,0,-1,0],[9E+09,0.0000,-275.7583,9E+09,9E+09,9E+09]];
	CONST robtarget p411:=[[0.0000,-167.6495,7.8481],[0.0000,-0.3314,0.9435,0.0000],[-1,0,-1,0],[9E+09,0.0000,-276.2869,9E+09,9E+09,9E+09]];
	CONST robtarget p412:=[[0.0000,-166.4077,7.8672],[0.0000,-0.3270,0.9450,0.0000],[-1,0,-1,0],[9E+09,0.0000,-276.8235,9E+09,9E+09,9E+09]];
	CONST robtarget p413:=[[0.0000,-165.1807,7.8863],[0.0000,-0.3225,0.9466,0.0000],[-1,0,-1,0],[9E+09,0.0000,-277.3681,9E+09,9E+09,9E+09]];
	CONST robtarget p414:=[[0.0000,-163.9689,7.9053],[0.0000,-0.3180,0.9481,0.0000],[-1,0,-1,0],[9E+09,0.0000,-277.9207,9E+09,9E+09,9E+09]];
	CONST robtarget p415:=[[0.0000,-162.7726,7.9244],[0.0000,-0.3133,0.9496,0.0000],[-1,0,-1,0],[9E+09,0.0000,-278.4816,9E+09,9E+09,9E+09]];
	CONST robtarget p416:=[[0.0000,-161.5921,7.9435],[0.0000,-0.3086,0.9512,0.0000],[-1,0,-1,0],[9E+09,0.0000,-279.0507,9E+09,9E+09,9E+09]];
	CONST robtarget p417:=[[0.0000,-160.4277,7.9626],[0.0000,-0.3038,0.9527,0.0000],[-1,0,-1,0],[9E+09,0.0000,-279.6282,9E+09,9E+09,9E+09]];
	CONST robtarget p418:=[[0.0000,-159.2799,7.9817],[0.0000,-0.2989,0.9543,0.0000],[-1,0,-1,0],[9E+09,0.0000,-280.2140,9E+09,9E+09,9E+09]];
	CONST robtarget p419:=[[0.0000,-158.1490,8.0008],[0.0000,-0.2940,0.9558,0.0000],[-1,0,-1,0],[9E+09,0.0000,-280.8082,9E+09,9E+09,9E+09]];
	CONST robtarget p420:=[[0.0000,-157.0354,8.0198],[0.0000,-0.2889,0.9573,0.0000],[-1,0,-1,0],[9E+09,0.0000,-281.4110,9E+09,9E+09,9E+09]];
	CONST robtarget p421:=[[0.0000,-155.9394,8.0389],[0.0000,-0.2838,0.9589,0.0000],[-1,0,-1,0],[9E+09,0.0000,-282.0223,9E+09,9E+09,9E+09]];
	CONST robtarget p422:=[[0.0000,-154.8613,8.0580],[0.0000,-0.2786,0.9604,0.0000],[-1,0,-1,0],[9E+09,0.0000,-282.6422,9E+09,9E+09,9E+09]];
	CONST robtarget p423:=[[0.0000,-153.8017,8.0771],[0.0000,-0.2734,0.9619,0.0000],[-1,0,-1,0],[9E+09,0.0000,-283.2706,9E+09,9E+09,9E+09]];
	CONST robtarget p424:=[[0.0000,-152.7608,8.0962],[0.0000,-0.2680,0.9634,0.0000],[-1,0,-1,0],[9E+09,0.0000,-283.9078,9E+09,9E+09,9E+09]];
	CONST robtarget p425:=[[0.0000,-151.7391,8.1153],[0.0000,-0.2626,0.9649,0.0000],[-1,0,-1,0],[9E+09,0.0000,-284.5536,9E+09,9E+09,9E+09]];
	CONST robtarget p426:=[[0.0000,-150.7369,8.1344],[0.0000,-0.2571,0.9664,0.0000],[-1,0,-1,0],[9E+09,0.0000,-285.2080,9E+09,9E+09,9E+09]];
	CONST robtarget p427:=[[0.0000,-149.7546,8.1534],[0.0000,-0.2515,0.9679,0.0000],[-1,0,-1,0],[9E+09,0.0000,-285.8712,9E+09,9E+09,9E+09]];
	CONST robtarget p428:=[[0.0000,-148.7927,8.1725],[0.0000,-0.2458,0.9693,0.0000],[-1,0,-1,0],[9E+09,0.0000,-286.5430,9E+09,9E+09,9E+09]];
	CONST robtarget p429:=[[0.0000,-147.8514,8.1916],[0.0000,-0.2400,0.9708,0.0000],[-1,0,-1,0],[9E+09,0.0000,-287.2234,9E+09,9E+09,9E+09]];
	CONST robtarget p430:=[[0.0000,-146.9313,8.2107],[0.0000,-0.2342,0.9722,0.0000],[-1,0,-1,0],[9E+09,0.0000,-287.9125,9E+09,9E+09,9E+09]];
	CONST robtarget p431:=[[0.0000,-146.0327,8.2298],[0.0000,-0.2283,0.9736,0.0000],[-1,0,-1,0],[9E+09,0.0000,-288.6102,9E+09,9E+09,9E+09]];
	CONST robtarget p432:=[[0.0000,-145.1561,8.2489],[0.0000,-0.2223,0.9750,0.0000],[-1,0,-1,0],[9E+09,0.0000,-289.3164,9E+09,9E+09,9E+09]];
	CONST robtarget p433:=[[0.0000,-144.3017,8.2679],[0.0000,-0.2162,0.9764,0.0000],[-1,0,-1,0],[9E+09,0.0000,-290.0310,9E+09,9E+09,9E+09]];
	CONST robtarget p434:=[[0.0000,-143.4701,8.2870],[0.0000,-0.2100,0.9777,0.0000],[-1,0,-1,0],[9E+09,0.0000,-290.7541,9E+09,9E+09,9E+09]];
	CONST robtarget p435:=[[0.0000,-142.6615,8.3061],[0.0000,-0.2038,0.9790,0.0000],[-1,0,-1,0],[9E+09,0.0000,-291.4854,9E+09,9E+09,9E+09]];
	CONST robtarget p436:=[[0.0000,-141.8765,8.3252],[0.0000,-0.1974,0.9803,0.0000],[-1,0,-1,0],[9E+09,0.0000,-292.2250,9E+09,9E+09,9E+09]];
	CONST robtarget p437:=[[0.0000,-141.1154,8.3443],[0.0000,-0.1910,0.9816,0.0000],[-1,0,-1,0],[9E+09,0.0000,-292.9727,9E+09,9E+09,9E+09]];
	CONST robtarget p438:=[[0.0000,-140.3786,8.3634],[0.0000,-0.1846,0.9828,0.0000],[-1,0,-1,0],[9E+09,0.0000,-293.7284,9E+09,9E+09,9E+09]];
	CONST robtarget p439:=[[0.0000,-139.6664,8.3824],[0.0000,-0.1780,0.9840,0.0000],[-1,0,-1,0],[9E+09,0.0000,-294.4919,9E+09,9E+09,9E+09]];
	CONST robtarget p440:=[[0.0000,-138.9793,8.4015],[0.0000,-0.1714,0.9852,0.0000],[-1,0,-1,0],[9E+09,0.0000,-295.2631,9E+09,9E+09,9E+09]];
	CONST robtarget p441:=[[0.0000,-138.3177,8.4206],[0.0000,-0.1647,0.9863,0.0000],[-1,0,-1,0],[9E+09,0.0000,-296.0418,9E+09,9E+09,9E+09]];
	CONST robtarget p442:=[[0.0000,-137.6818,8.4397],[0.0000,-0.1579,0.9875,0.0000],[-1,0,-1,0],[9E+09,0.0000,-296.8279,9E+09,9E+09,9E+09]];
	CONST robtarget p443:=[[0.0000,-137.0721,8.4588],[0.0000,-0.1511,0.9885,0.0000],[-1,0,-1,0],[9E+09,0.0000,-297.6211,9E+09,9E+09,9E+09]];
	CONST robtarget p444:=[[0.0000,-136.4888,8.4779],[0.0000,-0.1442,0.9896,0.0000],[-1,0,-1,0],[9E+09,0.0000,-298.4212,9E+09,9E+09,9E+09]];
	CONST robtarget p445:=[[0.0000,-135.9325,8.4969],[0.0000,-0.1372,0.9905,0.0000],[-1,0,-1,0],[9E+09,0.0000,-299.2281,9E+09,9E+09,9E+09]];
	CONST robtarget p446:=[[0.0000,-135.4032,8.5160],[0.0000,-0.1302,0.9915,0.0000],[-1,0,-1,0],[9E+09,0.0000,-300.0414,9E+09,9E+09,9E+09]];
	CONST robtarget p447:=[[0.0000,-134.9015,8.5351],[0.0000,-0.1231,0.9924,0.0000],[-1,0,-1,0],[9E+09,0.0000,-300.8609,9E+09,9E+09,9E+09]];
	CONST robtarget p448:=[[0.0000,-134.4276,8.5542],[0.0000,-0.1159,0.9933,0.0000],[-1,0,-1,0],[9E+09,0.0000,-301.6864,9E+09,9E+09,9E+09]];
	CONST robtarget p449:=[[0.0000,-133.9818,8.5733],[0.0000,-0.1087,0.9941,0.0000],[-1,0,-1,0],[9E+09,0.0000,-302.5175,9E+09,9E+09,9E+09]];
	CONST robtarget p450:=[[0.0000,-133.5644,8.5924],[0.0000,-0.1015,0.9948,0.0000],[-1,0,-1,0],[9E+09,0.0000,-303.3540,9E+09,9E+09,9E+09]];
	CONST robtarget p451:=[[0.0000,-133.1756,8.6115],[0.0000,-0.0941,0.9956,0.0000],[-1,0,-1,0],[9E+09,0.0000,-304.1956,9E+09,9E+09,9E+09]];
	CONST robtarget p452:=[[0.0000,-132.8157,8.6305],[0.0000,-0.0868,0.9962,0.0000],[-1,0,-1,0],[9E+09,0.0000,-305.0419,9E+09,9E+09,9E+09]];
	CONST robtarget p453:=[[0.0000,-132.4849,8.6496],[0.0000,-0.0794,0.9968,0.0000],[-1,0,-1,0],[9E+09,0.0000,-305.8927,9E+09,9E+09,9E+09]];
	CONST robtarget p454:=[[0.0000,-132.1835,8.6687],[0.0000,-0.0720,0.9974,0.0000],[-1,0,-1,0],[9E+09,0.0000,-306.7475,9E+09,9E+09,9E+09]];
	CONST robtarget p455:=[[0.0000,-131.9116,8.6878],[0.0000,-0.0645,0.9979,0.0000],[-1,0,-1,0],[9E+09,0.0000,-307.6060,9E+09,9E+09,9E+09]];
	CONST robtarget p456:=[[0.0000,-131.6695,8.7069],[0.0000,-0.0570,0.9984,0.0000],[-1,0,-1,0],[9E+09,0.0000,-308.4679,9E+09,9E+09,9E+09]];
	CONST robtarget p457:=[[0.0000,-131.4573,8.7260],[0.0000,-0.0494,0.9988,0.0000],[-1,0,-1,0],[9E+09,0.0000,-309.3327,9E+09,9E+09,9E+09]];
	CONST robtarget p458:=[[0.0000,-131.2751,8.7450],[0.0000,-0.0419,0.9991,0.0000],[-1,0,-1,0],[9E+09,0.0000,-310.2002,9E+09,9E+09,9E+09]];
	CONST robtarget p459:=[[0.0000,-131.1231,8.7641],[0.0000,-0.0343,0.9994,0.0000],[-1,0,-1,0],[9E+09,0.0000,-311.0698,9E+09,9E+09,9E+09]];
	CONST robtarget p460:=[[0.0000,-131.0014,8.7832],[0.0000,-0.0267,0.9996,0.0000],[-1,0,-1,0],[9E+09,0.0000,-311.9413,9E+09,9E+09,9E+09]];
	CONST robtarget p461:=[[0.0000,-130.9100,8.8023],[0.0000,-0.0191,0.9998,0.0000],[-1,0,-1,0],[9E+09,0.0000,-312.8142,9E+09,9E+09,9E+09]];
	CONST robtarget p462:=[[0.0000,-130.8491,8.8214],[0.0000,-0.0114,0.9999,0.0000],[-1,0,-1,0],[9E+09,0.0000,-313.6881,9E+09,9E+09,9E+09]];
	CONST robtarget p463:=[[0.0000,-130.8186,8.8405],[0.0000,-0.0038,1.0000,0.0000],[-1,0,-1,0],[9E+09,0.0000,-314.5626,9E+09,9E+09,9E+09]];
	CONST robtarget p464:=[[0.0000,-130.8186,8.8595],[0.0000,-0.0038,-1.0000,0.0000],[-1,0,-1,0],[9E+09,0.0000,-315.4374,9E+09,9E+09,9E+09]];
	CONST robtarget p465:=[[0.0000,-130.8491,8.8786],[0.0000,-0.0114,-0.9999,0.0000],[-1,0,-1,0],[9E+09,0.0000,-316.3119,9E+09,9E+09,9E+09]];
	CONST robtarget p466:=[[0.0000,-130.9100,8.8977],[0.0000,-0.0191,-0.9998,0.0000],[-1,0,-1,0],[9E+09,0.0000,-317.1858,9E+09,9E+09,9E+09]];
	CONST robtarget p467:=[[0.0000,-131.0014,8.9168],[0.0000,-0.0267,-0.9996,0.0000],[-1,0,-1,0],[9E+09,0.0000,-318.0587,9E+09,9E+09,9E+09]];
	CONST robtarget p468:=[[0.0000,-131.1231,8.9359],[0.0000,-0.0343,-0.9994,0.0000],[-1,0,-1,0],[9E+09,0.0000,-318.9302,9E+09,9E+09,9E+09]];
	CONST robtarget p469:=[[0.0000,-131.2751,8.9550],[0.0000,-0.0419,-0.9991,0.0000],[-1,0,-1,0],[9E+09,0.0000,-319.7998,9E+09,9E+09,9E+09]];
	CONST robtarget p470:=[[0.0000,-131.4573,8.9740],[0.0000,-0.0494,-0.9988,0.0000],[-1,0,-1,0],[9E+09,0.0000,-320.6673,9E+09,9E+09,9E+09]];
	CONST robtarget p471:=[[0.0000,-131.6695,8.9931],[0.0000,-0.0570,-0.9984,0.0000],[-1,0,-1,0],[9E+09,0.0000,-321.5321,9E+09,9E+09,9E+09]];
	CONST robtarget p472:=[[0.0000,-131.9116,9.0122],[0.0000,-0.0645,-0.9979,0.0000],[-1,0,-1,0],[9E+09,0.0000,-322.3940,9E+09,9E+09,9E+09]];
	CONST robtarget p473:=[[0.0000,-132.1835,9.0313],[0.0000,-0.0720,-0.9974,0.0000],[-1,0,-1,0],[9E+09,0.0000,-323.2525,9E+09,9E+09,9E+09]];
	CONST robtarget p474:=[[0.0000,-132.4849,9.0504],[0.0000,-0.0794,-0.9968,0.0000],[-1,0,-1,0],[9E+09,0.0000,-324.1073,9E+09,9E+09,9E+09]];
	CONST robtarget p475:=[[0.0000,-132.8157,9.0695],[0.0000,-0.0868,-0.9962,0.0000],[-1,0,-1,0],[9E+09,0.0000,-324.9581,9E+09,9E+09,9E+09]];
	CONST robtarget p476:=[[0.0000,-133.1756,9.0885],[0.0000,-0.0941,-0.9956,0.0000],[-1,0,-1,0],[9E+09,0.0000,-325.8044,9E+09,9E+09,9E+09]];
	CONST robtarget p477:=[[0.0000,-133.5644,9.1076],[0.0000,-0.1015,-0.9948,0.0000],[-1,0,-1,0],[9E+09,0.0000,-326.6460,9E+09,9E+09,9E+09]];
	CONST robtarget p478:=[[0.0000,-133.9818,9.1267],[0.0000,-0.1087,-0.9941,0.0000],[-1,0,-1,0],[9E+09,0.0000,-327.4825,9E+09,9E+09,9E+09]];
	CONST robtarget p479:=[[0.0000,-134.4276,9.1458],[0.0000,-0.1159,-0.9933,0.0000],[-1,0,-1,0],[9E+09,0.0000,-328.3136,9E+09,9E+09,9E+09]];
	CONST robtarget p480:=[[0.0000,-134.9015,9.1649],[0.0000,-0.1231,-0.9924,0.0000],[-1,0,-1,0],[9E+09,0.0000,-329.1391,9E+09,9E+09,9E+09]];
	CONST robtarget p481:=[[0.0000,-135.4032,9.1840],[0.0000,-0.1302,-0.9915,0.0000],[-1,0,-1,0],[9E+09,0.0000,-329.9586,9E+09,9E+09,9E+09]];
	CONST robtarget p482:=[[0.0000,-135.9325,9.2031],[0.0000,-0.1372,-0.9905,0.0000],[-1,0,-1,0],[9E+09,0.0000,-330.7719,9E+09,9E+09,9E+09]];
	CONST robtarget p483:=[[0.0000,-136.4888,9.2221],[0.0000,-0.1442,-0.9896,0.0000],[-1,0,-1,0],[9E+09,0.0000,-331.5788,9E+09,9E+09,9E+09]];
	CONST robtarget p484:=[[0.0000,-137.0721,9.2412],[0.0000,-0.1511,-0.9885,0.0000],[-1,0,-1,0],[9E+09,0.0000,-332.3789,9E+09,9E+09,9E+09]];
	CONST robtarget p485:=[[0.0000,-137.6818,9.2603],[0.0000,-0.1579,-0.9875,0.0000],[-1,0,-1,0],[9E+09,0.0000,-333.1721,9E+09,9E+09,9E+09]];
	CONST robtarget p486:=[[0.0000,-138.3177,9.2794],[0.0000,-0.1647,-0.9863,0.0000],[-1,0,-1,0],[9E+09,0.0000,-333.9582,9E+09,9E+09,9E+09]];
	CONST robtarget p487:=[[0.0000,-138.9793,9.2985],[0.0000,-0.1714,-0.9852,0.0000],[-1,0,-1,0],[9E+09,0.0000,-334.7369,9E+09,9E+09,9E+09]];
	CONST robtarget p488:=[[0.0000,-139.6664,9.3176],[0.0000,-0.1780,-0.9840,0.0000],[-1,0,-1,0],[9E+09,0.0000,-335.5081,9E+09,9E+09,9E+09]];
	CONST robtarget p489:=[[0.0000,-140.3786,9.3366],[0.0000,-0.1846,-0.9828,0.0000],[-1,0,-1,0],[9E+09,0.0000,-336.2716,9E+09,9E+09,9E+09]];
	CONST robtarget p490:=[[0.0000,-141.1154,9.3557],[0.0000,-0.1910,-0.9816,0.0000],[-1,0,-1,0],[9E+09,0.0000,-337.0273,9E+09,9E+09,9E+09]];
	CONST robtarget p491:=[[0.0000,-141.8765,9.3748],[0.0000,-0.1974,-0.9803,0.0000],[-1,0,-1,0],[9E+09,0.0000,-337.7750,9E+09,9E+09,9E+09]];
	CONST robtarget p492:=[[0.0000,-142.6615,9.3939],[0.0000,-0.2038,-0.9790,0.0000],[-1,0,-1,0],[9E+09,0.0000,-338.5146,9E+09,9E+09,9E+09]];
	CONST robtarget p493:=[[0.0000,-143.4701,9.4130],[0.0000,-0.2100,-0.9777,0.0000],[-1,0,-1,0],[9E+09,0.0000,-339.2459,9E+09,9E+09,9E+09]];
	CONST robtarget p494:=[[0.0000,-144.3017,9.4321],[0.0000,-0.2162,-0.9764,0.0000],[-1,0,-1,0],[9E+09,0.0000,-339.9690,9E+09,9E+09,9E+09]];
	CONST robtarget p495:=[[0.0000,-145.1561,9.4511],[0.0000,-0.2223,-0.9750,0.0000],[-1,0,-1,0],[9E+09,0.0000,-340.6836,9E+09,9E+09,9E+09]];
	CONST robtarget p496:=[[0.0000,-146.0327,9.4702],[0.0000,-0.2283,-0.9736,0.0000],[-1,0,-1,0],[9E+09,0.0000,-341.3898,9E+09,9E+09,9E+09]];
	CONST robtarget p497:=[[0.0000,-146.9313,9.4893],[0.0000,-0.2342,-0.9722,0.0000],[-1,0,-1,0],[9E+09,0.0000,-342.0875,9E+09,9E+09,9E+09]];
	CONST robtarget p498:=[[0.0000,-147.8514,9.5084],[0.0000,-0.2400,-0.9708,0.0000],[-1,0,-1,0],[9E+09,0.0000,-342.7766,9E+09,9E+09,9E+09]];
	CONST robtarget p499:=[[0.0000,-148.7927,9.5275],[0.0000,-0.2458,-0.9693,0.0000],[-1,0,-1,0],[9E+09,0.0000,-343.4570,9E+09,9E+09,9E+09]];
	CONST robtarget p500:=[[0.0000,-149.7546,9.5466],[0.0000,-0.2515,-0.9679,0.0000],[-1,0,-1,0],[9E+09,0.0000,-344.1288,9E+09,9E+09,9E+09]];
	CONST robtarget p501:=[[0.0000,-150.7369,9.5656],[0.0000,-0.2571,-0.9664,0.0000],[-1,0,-1,0],[9E+09,0.0000,-344.7920,9E+09,9E+09,9E+09]];
	CONST robtarget p502:=[[0.0000,-151.7391,9.5847],[0.0000,-0.2626,-0.9649,0.0000],[-1,0,-1,0],[9E+09,0.0000,-345.4464,9E+09,9E+09,9E+09]];
	CONST robtarget p503:=[[0.0000,-152.7608,9.6038],[0.0000,-0.2680,-0.9634,0.0000],[-1,0,-1,0],[9E+09,0.0000,-346.0922,9E+09,9E+09,9E+09]];
	CONST robtarget p504:=[[0.0000,-153.8017,9.6229],[0.0000,-0.2734,-0.9619,0.0000],[-1,0,-1,0],[9E+09,0.0000,-346.7294,9E+09,9E+09,9E+09]];
	CONST robtarget p505:=[[0.0000,-154.8613,9.6420],[0.0000,-0.2786,-0.9604,0.0000],[-1,0,-1,0],[9E+09,0.0000,-347.3578,9E+09,9E+09,9E+09]];
	CONST robtarget p506:=[[0.0000,-155.9394,9.6611],[0.0000,-0.2838,-0.9589,0.0000],[-1,0,-1,0],[9E+09,0.0000,-347.9777,9E+09,9E+09,9E+09]];
	CONST robtarget p507:=[[0.0000,-157.0354,9.6802],[0.0000,-0.2889,-0.9573,0.0000],[-1,0,-1,0],[9E+09,0.0000,-348.5890,9E+09,9E+09,9E+09]];
	CONST robtarget p508:=[[0.0000,-158.1490,9.6992],[0.0000,-0.2940,-0.9558,0.0000],[-1,0,-1,0],[9E+09,0.0000,-349.1918,9E+09,9E+09,9E+09]];
	CONST robtarget p509:=[[0.0000,-159.2799,9.7183],[0.0000,-0.2989,-0.9543,0.0000],[-1,0,-1,0],[9E+09,0.0000,-349.7860,9E+09,9E+09,9E+09]];
	CONST robtarget p510:=[[0.0000,-160.4277,9.7374],[0.0000,-0.3038,-0.9527,0.0000],[-1,0,-1,0],[9E+09,0.0000,-350.3718,9E+09,9E+09,9E+09]];
	CONST robtarget p511:=[[0.0000,-161.5921,9.7565],[0.0000,-0.3086,-0.9512,0.0000],[-1,0,-1,0],[9E+09,0.0000,-350.9493,9E+09,9E+09,9E+09]];
	CONST robtarget p512:=[[0.0000,-162.7726,9.7756],[0.0000,-0.3133,-0.9496,0.0000],[-1,0,-1,0],[9E+09,0.0000,-351.5184,9E+09,9E+09,9E+09]];
	CONST robtarget p513:=[[0.0000,-163.9689,9.7947],[0.0000,-0.3180,-0.9481,0.0000],[-1,0,-1,0],[9E+09,0.0000,-352.0793,9E+09,9E+09,9E+09]];
	CONST robtarget p514:=[[0.0000,-165.1807,9.8137],[0.0000,-0.3225,-0.9466,0.0000],[-1,0,-1,0],[9E+09,0.0000,-352.6319,9E+09,9E+09,9E+09]];
	CONST robtarget p515:=[[0.0000,-166.4077,9.8328],[0.0000,-0.3270,-0.9450,0.0000],[-1,0,-1,0],[9E+09,0.0000,-353.1765,9E+09,9E+09,9E+09]];
	CONST robtarget p516:=[[0.0000,-167.6495,9.8519],[0.0000,-0.3314,-0.9435,0.0000],[-1,0,-1,0],[9E+09,0.0000,-353.7131,9E+09,9E+09,9E+09]];
	CONST robtarget p517:=[[0.0000,-168.9057,9.8710],[0.0000,-0.3358,-0.9419,0.0000],[-1,0,-1,0],[9E+09,0.0000,-354.2417,9E+09,9E+09,9E+09]];
	CONST robtarget p518:=[[0.0000,-170.1762,9.8901],[0.0000,-0.3401,-0.9404,0.0000],[-1,0,-1,0],[9E+09,0.0000,-354.7625,9E+09,9E+09,9E+09]];
	CONST robtarget p519:=[[0.0000,-171.4604,9.9092],[0.0000,-0.3443,-0.9389,0.0000],[-1,0,-1,0],[9E+09,0.0000,-355.2755,9E+09,9E+09,9E+09]];
	CONST robtarget p520:=[[0.0000,-172.7582,9.9282],[0.0000,-0.3484,-0.9373,0.0000],[-1,0,-1,0],[9E+09,0.0000,-355.7809,9E+09,9E+09,9E+09]];
	CONST robtarget p521:=[[0.0000,-174.0693,9.9473],[0.0000,-0.3525,-0.9358,0.0000],[-1,0,-1,0],[9E+09,0.0000,-356.2787,9E+09,9E+09,9E+09]];
	CONST robtarget p522:=[[0.0000,-175.3933,9.9664],[0.0000,-0.3565,-0.9343,0.0000],[-1,0,-1,0],[9E+09,0.0000,-356.7690,9E+09,9E+09,9E+09]];
	CONST robtarget p523:=[[0.0000,-176.7300,9.9855],[0.0000,-0.3604,-0.9328,0.0000],[-1,0,-1,0],[9E+09,0.0000,-357.2519,9E+09,9E+09,9E+09]];
	CONST robtarget p524:=[[0.0000,-178.0790,10.0046],[0.0000,-0.3643,-0.9313,0.0000],[-1,0,-1,0],[9E+09,0.0000,-357.7276,9E+09,9E+09,9E+09]];
	CONST robtarget p525:=[[0.0000,-179.4401,10.0237],[0.0000,-0.3681,-0.9298,0.0000],[-1,0,-1,0],[9E+09,0.0000,-358.1960,9E+09,9E+09,9E+09]];
	CONST robtarget p526:=[[0.0000,-180.8130,10.0427],[0.0000,-0.3718,-0.9283,0.0000],[-1,0,-1,0],[9E+09,0.0000,-358.6574,9E+09,9E+09,9E+09]];
	CONST robtarget p527:=[[0.0000,-182.1975,10.0618],[0.0000,-0.3755,-0.9268,0.0000],[-1,0,-1,0],[9E+09,0.0000,-359.1118,9E+09,9E+09,9E+09]];
	CONST robtarget p528:=[[0.0000,-183.5932,10.0809],[0.0000,-0.3791,-0.9253,0.0000],[-1,0,-1,0],[9E+09,0.0000,-359.5593,9E+09,9E+09,9E+09]];
	CONST robtarget p529:=[[0.0000,-185.0000,10.1000],[0.0000,-0.3890,0.9212,0.0000],[-1,0,-1,0],[9E+09,0.0000,-360.0000,9E+09,9E+09,9E+09]];
	CONST robtarget p530:=[[0.0000,-183.5821,10.1192],[0.0000,-0.3855,0.9227,0.0000],[-1,0,-1,0],[9E+09,0.0000,-360.4321,9E+09,9E+09,9E+09]];
	CONST robtarget p531:=[[0.0000,-182.1749,10.1385],[0.0000,-0.3820,0.9242,0.0000],[-1,0,-1,0],[9E+09,0.0000,-360.8710,9E+09,9E+09,9E+09]];
	CONST robtarget p532:=[[0.0000,-180.7785,10.1577],[0.0000,-0.3784,0.9256,0.0000],[-1,0,-1,0],[9E+09,0.0000,-361.3166,9E+09,9E+09,9E+09]];
	CONST robtarget p533:=[[0.0000,-179.3932,10.1769],[0.0000,-0.3747,0.9271,0.0000],[-1,0,-1,0],[9E+09,0.0000,-361.7692,9E+09,9E+09,9E+09]];
	CONST robtarget p534:=[[0.0000,-178.0193,10.1962],[0.0000,-0.3710,0.9286,0.0000],[-1,0,-1,0],[9E+09,0.0000,-362.2288,9E+09,9E+09,9E+09]];
	CONST robtarget p535:=[[0.0000,-176.6570,10.2154],[0.0000,-0.3672,0.9301,0.0000],[-1,0,-1,0],[9E+09,0.0000,-362.6955,9E+09,9E+09,9E+09]];
	CONST robtarget p536:=[[0.0000,-175.3066,10.2346],[0.0000,-0.3634,0.9316,0.0000],[-1,0,-1,0],[9E+09,0.0000,-363.1694,9E+09,9E+09,9E+09]];
	CONST robtarget p537:=[[0.0000,-173.9684,10.2538],[0.0000,-0.3595,0.9332,0.0000],[-1,0,-1,0],[9E+09,0.0000,-363.6506,9E+09,9E+09,9E+09]];
	CONST robtarget p538:=[[0.0000,-172.6426,10.2731],[0.0000,-0.3555,0.9347,0.0000],[-1,0,-1,0],[9E+09,0.0000,-364.1393,9E+09,9E+09,9E+09]];
	CONST robtarget p539:=[[0.0000,-171.3296,10.2923],[0.0000,-0.3514,0.9362,0.0000],[-1,0,-1,0],[9E+09,0.0000,-364.6355,9E+09,9E+09,9E+09]];
	CONST robtarget p540:=[[0.0000,-170.0297,10.3115],[0.0000,-0.3473,0.9378,0.0000],[-1,0,-1,0],[9E+09,0.0000,-365.1393,9E+09,9E+09,9E+09]];
	CONST robtarget p541:=[[0.0000,-168.7431,10.3308],[0.0000,-0.3431,0.9393,0.0000],[-1,0,-1,0],[9E+09,0.0000,-365.6508,9E+09,9E+09,9E+09]];
	CONST robtarget p542:=[[0.0000,-167.4701,10.3500],[0.0000,-0.3389,0.9408,0.0000],[-1,0,-1,0],[9E+09,0.0000,-366.1702,9E+09,9E+09,9E+09]];
	CONST robtarget p543:=[[0.0000,-166.2112,10.3692],[0.0000,-0.3345,0.9424,0.0000],[-1,0,-1,0],[9E+09,0.0000,-366.6974,9E+09,9E+09,9E+09]];
	CONST robtarget p544:=[[0.0000,-164.9665,10.3885],[0.0000,-0.3301,0.9439,0.0000],[-1,0,-1,0],[9E+09,0.0000,-367.2327,9E+09,9E+09,9E+09]];
	CONST robtarget p545:=[[0.0000,-163.7364,10.4077],[0.0000,-0.3256,0.9455,0.0000],[-1,0,-1,0],[9E+09,0.0000,-367.7761,9E+09,9E+09,9E+09]];
	CONST robtarget p546:=[[0.0000,-162.5213,10.4269],[0.0000,-0.3211,0.9471,0.0000],[-1,0,-1,0],[9E+09,0.0000,-368.3276,9E+09,9E+09,9E+09]];
	CONST robtarget p547:=[[0.0000,-161.3215,10.4462],[0.0000,-0.3165,0.9486,0.0000],[-1,0,-1,0],[9E+09,0.0000,-368.8874,9E+09,9E+09,9E+09]];
	CONST robtarget p548:=[[0.0000,-160.1373,10.4654],[0.0000,-0.3117,0.9502,0.0000],[-1,0,-1,0],[9E+09,0.0000,-369.4555,9E+09,9E+09,9E+09]];
	CONST robtarget p549:=[[0.0000,-158.9690,10.4846],[0.0000,-0.3070,0.9517,0.0000],[-1,0,-1,0],[9E+09,0.0000,-370.0321,9E+09,9E+09,9E+09]];
	CONST robtarget p550:=[[0.0000,-157.8171,10.5038],[0.0000,-0.3021,0.9533,0.0000],[-1,0,-1,0],[9E+09,0.0000,-370.6171,9E+09,9E+09,9E+09]];
	CONST robtarget p551:=[[0.0000,-156.6819,10.5231],[0.0000,-0.2972,0.9548,0.0000],[-1,0,-1,0],[9E+09,0.0000,-371.2106,9E+09,9E+09,9E+09]];
	CONST robtarget p552:=[[0.0000,-155.5638,10.5423],[0.0000,-0.2921,0.9564,0.0000],[-1,0,-1,0],[9E+09,0.0000,-371.8128,9E+09,9E+09,9E+09]];
	CONST robtarget p553:=[[0.0000,-154.4631,10.5615],[0.0000,-0.2870,0.9579,0.0000],[-1,0,-1,0],[9E+09,0.0000,-372.4236,9E+09,9E+09,9E+09]];
	CONST robtarget p554:=[[0.0000,-153.3802,10.5808],[0.0000,-0.2819,0.9595,0.0000],[-1,0,-1,0],[9E+09,0.0000,-373.0431,9E+09,9E+09,9E+09]];
	CONST robtarget p555:=[[0.0000,-152.3155,10.6000],[0.0000,-0.2766,0.9610,0.0000],[-1,0,-1,0],[9E+09,0.0000,-373.6713,9E+09,9E+09,9E+09]];
	CONST robtarget p556:=[[0.0000,-151.2693,10.6192],[0.0000,-0.2712,0.9625,0.0000],[-1,0,-1,0],[9E+09,0.0000,-374.3083,9E+09,9E+09,9E+09]];
	CONST robtarget p557:=[[0.0000,-150.2421,10.6385],[0.0000,-0.2658,0.9640,0.0000],[-1,0,-1,0],[9E+09,0.0000,-374.9541,9E+09,9E+09,9E+09]];
	CONST robtarget p558:=[[0.0000,-149.2343,10.6577],[0.0000,-0.2603,0.9655,0.0000],[-1,0,-1,0],[9E+09,0.0000,-375.6087,9E+09,9E+09,9E+09]];
	CONST robtarget p559:=[[0.0000,-148.2462,10.6769],[0.0000,-0.2547,0.9670,0.0000],[-1,0,-1,0],[9E+09,0.0000,-376.2721,9E+09,9E+09,9E+09]];
	CONST robtarget p560:=[[0.0000,-147.2782,10.6962],[0.0000,-0.2490,0.9685,0.0000],[-1,0,-1,0],[9E+09,0.0000,-376.9443,9E+09,9E+09,9E+09]];
	CONST robtarget p561:=[[0.0000,-146.3308,10.7154],[0.0000,-0.2433,0.9700,0.0000],[-1,0,-1,0],[9E+09,0.0000,-377.6253,9E+09,9E+09,9E+09]];
	CONST robtarget p562:=[[0.0000,-145.4043,10.7346],[0.0000,-0.2374,0.9714,0.0000],[-1,0,-1,0],[9E+09,0.0000,-378.3151,9E+09,9E+09,9E+09]];
	CONST robtarget p563:=[[0.0000,-144.4991,10.7538],[0.0000,-0.2315,0.9728,0.0000],[-1,0,-1,0],[9E+09,0.0000,-379.0137,9E+09,9E+09,9E+09]];
	CONST robtarget p564:=[[0.0000,-143.6157,10.7731],[0.0000,-0.2255,0.9742,0.0000],[-1,0,-1,0],[9E+09,0.0000,-379.7209,9E+09,9E+09,9E+09]];
	CONST robtarget p565:=[[0.0000,-142.7545,10.7923],[0.0000,-0.2194,0.9756,0.0000],[-1,0,-1,0],[9E+09,0.0000,-380.4368,9E+09,9E+09,9E+09]];
	CONST robtarget p566:=[[0.0000,-141.9158,10.8115],[0.0000,-0.2132,0.9770,0.0000],[-1,0,-1,0],[9E+09,0.0000,-381.1613,9E+09,9E+09,9E+09]];
	CONST robtarget p567:=[[0.0000,-141.1001,10.8308],[0.0000,-0.2070,0.9783,0.0000],[-1,0,-1,0],[9E+09,0.0000,-381.8942,9E+09,9E+09,9E+09]];
	CONST robtarget p568:=[[0.0000,-140.3077,10.8500],[0.0000,-0.2006,0.9797,0.0000],[-1,0,-1,0],[9E+09,0.0000,-382.6356,9E+09,9E+09,9E+09]];
	CONST robtarget p569:=[[0.0000,-139.5391,10.8692],[0.0000,-0.1942,0.9810,0.0000],[-1,0,-1,0],[9E+09,0.0000,-383.3852,9E+09,9E+09,9E+09]];
	CONST robtarget p570:=[[0.0000,-138.7946,10.8885],[0.0000,-0.1877,0.9822,0.0000],[-1,0,-1,0],[9E+09,0.0000,-384.1430,9E+09,9E+09,9E+09]];
	CONST robtarget p571:=[[0.0000,-138.0747,10.9077],[0.0000,-0.1812,0.9835,0.0000],[-1,0,-1,0],[9E+09,0.0000,-384.9089,9E+09,9E+09,9E+09]];
	CONST robtarget p572:=[[0.0000,-137.3797,10.9269],[0.0000,-0.1745,0.9847,0.0000],[-1,0,-1,0],[9E+09,0.0000,-385.6827,9E+09,9E+09,9E+09]];
	CONST robtarget p573:=[[0.0000,-136.7100,10.9462],[0.0000,-0.1678,0.9858,0.0000],[-1,0,-1,0],[9E+09,0.0000,-386.4641,9E+09,9E+09,9E+09]];
	CONST robtarget p574:=[[0.0000,-136.0659,10.9654],[0.0000,-0.1610,0.9870,0.0000],[-1,0,-1,0],[9E+09,0.0000,-387.2531,9E+09,9E+09,9E+09]];
	CONST robtarget p575:=[[0.0000,-135.4480,10.9846],[0.0000,-0.1542,0.9880,0.0000],[-1,0,-1,0],[9E+09,0.0000,-388.0495,9E+09,9E+09,9E+09]];
	CONST robtarget p576:=[[0.0000,-134.8564,11.0038],[0.0000,-0.1472,0.9891,0.0000],[-1,0,-1,0],[9E+09,0.0000,-388.8530,9E+09,9E+09,9E+09]];
	CONST robtarget p577:=[[0.0000,-134.2916,11.0231],[0.0000,-0.1402,0.9901,0.0000],[-1,0,-1,0],[9E+09,0.0000,-389.6635,9E+09,9E+09,9E+09]];
	CONST robtarget p578:=[[0.0000,-133.7539,11.0423],[0.0000,-0.1332,0.9911,0.0000],[-1,0,-1,0],[9E+09,0.0000,-390.4806,9E+09,9E+09,9E+09]];
	CONST robtarget p579:=[[0.0000,-133.2436,11.0615],[0.0000,-0.1260,0.9920,0.0000],[-1,0,-1,0],[9E+09,0.0000,-391.3041,9E+09,9E+09,9E+09]];
	CONST robtarget p580:=[[0.0000,-132.7610,11.0808],[0.0000,-0.1188,0.9929,0.0000],[-1,0,-1,0],[9E+09,0.0000,-392.1338,9E+09,9E+09,9E+09]];
	CONST robtarget p581:=[[0.0000,-132.3065,11.1000],[0.0000,-0.1116,0.9938,0.0000],[-1,0,-1,0],[9E+09,0.0000,-392.9694,9E+09,9E+09,9E+09]];
	CONST robtarget p582:=[[0.0000,-131.8803,11.1192],[0.0000,-0.1043,0.9945,0.0000],[-1,0,-1,0],[9E+09,0.0000,-393.8106,9E+09,9E+09,9E+09]];
	CONST robtarget p583:=[[0.0000,-131.4827,11.1385],[0.0000,-0.0970,0.9953,0.0000],[-1,0,-1,0],[9E+09,0.0000,-394.6570,9E+09,9E+09,9E+09]];
	CONST robtarget p584:=[[0.0000,-131.1139,11.1577],[0.0000,-0.0896,0.9960,0.0000],[-1,0,-1,0],[9E+09,0.0000,-395.5084,9E+09,9E+09,9E+09]];
	CONST robtarget p585:=[[0.0000,-130.7743,11.1769],[0.0000,-0.0821,0.9966,0.0000],[-1,0,-1,0],[9E+09,0.0000,-396.3644,9E+09,9E+09,9E+09]];
	CONST robtarget p586:=[[0.0000,-130.4640,11.1962],[0.0000,-0.0746,0.9972,0.0000],[-1,0,-1,0],[9E+09,0.0000,-397.2246,9E+09,9E+09,9E+09]];
	CONST robtarget p587:=[[0.0000,-130.1833,11.2154],[0.0000,-0.0671,0.9977,0.0000],[-1,0,-1,0],[9E+09,0.0000,-398.0888,9E+09,9E+09,9E+09]];
	CONST robtarget p588:=[[0.0000,-129.9323,11.2346],[0.0000,-0.0596,0.9982,0.0000],[-1,0,-1,0],[9E+09,0.0000,-398.9565,9E+09,9E+09,9E+09]];
	CONST robtarget p589:=[[0.0000,-129.7112,11.2538],[0.0000,-0.0520,0.9986,0.0000],[-1,0,-1,0],[9E+09,0.0000,-399.8273,9E+09,9E+09,9E+09]];
	CONST robtarget p590:=[[0.0000,-129.5202,11.2731],[0.0000,-0.0444,0.9990,0.0000],[-1,0,-1,0],[9E+09,0.0000,-400.7009,9E+09,9E+09,9E+09]];
	CONST robtarget p591:=[[0.0000,-129.3594,11.2923],[0.0000,-0.0367,0.9993,0.0000],[-1,0,-1,0],[9E+09,0.0000,-401.5770,9E+09,9E+09,9E+09]];
	CONST robtarget p592:=[[0.0000,-129.2289,11.3115],[0.0000,-0.0291,0.9996,0.0000],[-1,0,-1,0],[9E+09,0.0000,-402.4549,9E+09,9E+09,9E+09]];
	CONST robtarget p593:=[[0.0000,-129.1287,11.3308],[0.0000,-0.0214,0.9998,0.0000],[-1,0,-1,0],[9E+09,0.0000,-403.3345,9E+09,9E+09,9E+09]];
	CONST robtarget p594:=[[0.0000,-129.0591,11.3500],[0.0000,-0.0137,0.9999,0.0000],[-1,0,-1,0],[9E+09,0.0000,-404.2152,9E+09,9E+09,9E+09]];
	CONST robtarget p595:=[[0.0000,-129.0200,11.3692],[0.0000,-0.0060,1.0000,0.0000],[-1,0,-1,0],[9E+09,0.0000,-405.0966,9E+09,9E+09,9E+09]];
	CONST robtarget p596:=[[0.0000,-129.0114,11.3885],[0.0000,-0.0017,-1.0000,0.0000],[-1,0,-1,0],[9E+09,0.0000,-405.9784,9E+09,9E+09,9E+09]];
	CONST robtarget p597:=[[0.0000,-129.0334,11.4077],[0.0000,-0.0094,-1.0000,0.0000],[-1,0,-1,0],[9E+09,0.0000,-406.8601,9E+09,9E+09,9E+09]];
	CONST robtarget p598:=[[0.0000,-129.0859,11.4269],[0.0000,-0.0171,-0.9999,0.0000],[-1,0,-1,0],[9E+09,0.0000,-407.7412,9E+09,9E+09,9E+09]];
	CONST robtarget p599:=[[0.0000,-129.1689,11.4462],[0.0000,-0.0248,-0.9997,0.0000],[-1,0,-1,0],[9E+09,0.0000,-408.6215,9E+09,9E+09,9E+09]];
	CONST robtarget p600:=[[0.0000,-129.2824,11.4654],[0.0000,-0.0324,-0.9995,0.0000],[-1,0,-1,0],[9E+09,0.0000,-409.5004,9E+09,9E+09,9E+09]];
	CONST robtarget p601:=[[0.0000,-129.4262,11.4846],[0.0000,-0.0401,-0.9992,0.0000],[-1,0,-1,0],[9E+09,0.0000,-410.3776,9E+09,9E+09,9E+09]];
	CONST robtarget p602:=[[0.0000,-129.6003,11.5038],[0.0000,-0.0477,-0.9989,0.0000],[-1,0,-1,0],[9E+09,0.0000,-411.2526,9E+09,9E+09,9E+09]];
	CONST robtarget p603:=[[0.0000,-129.8046,11.5231],[0.0000,-0.0553,-0.9985,0.0000],[-1,0,-1,0],[9E+09,0.0000,-412.1250,9E+09,9E+09,9E+09]];
	CONST robtarget p604:=[[0.0000,-130.0388,11.5423],[0.0000,-0.0629,-0.9980,0.0000],[-1,0,-1,0],[9E+09,0.0000,-412.9945,9E+09,9E+09,9E+09]];
	CONST robtarget p605:=[[0.0000,-130.3029,11.5615],[0.0000,-0.0704,-0.9975,0.0000],[-1,0,-1,0],[9E+09,0.0000,-413.8607,9E+09,9E+09,9E+09]];
	CONST robtarget p606:=[[0.0000,-130.5966,11.5808],[0.0000,-0.0779,-0.9970,0.0000],[-1,0,-1,0],[9E+09,0.0000,-414.7232,9E+09,9E+09,9E+09]];
	CONST robtarget p607:=[[0.0000,-130.9198,11.6000],[0.0000,-0.0854,-0.9963,0.0000],[-1,0,-1,0],[9E+09,0.0000,-415.5816,9E+09,9E+09,9E+09]];
	CONST robtarget p608:=[[0.0000,-131.2723,11.6192],[0.0000,-0.0928,-0.9957,0.0000],[-1,0,-1,0],[9E+09,0.0000,-416.4356,9E+09,9E+09,9E+09]];
	CONST robtarget p609:=[[0.0000,-131.6537,11.6385],[0.0000,-0.1002,-0.9950,0.0000],[-1,0,-1,0],[9E+09,0.0000,-417.2849,9E+09,9E+09,9E+09]];
	CONST robtarget p610:=[[0.0000,-132.0639,11.6577],[0.0000,-0.1075,-0.9942,0.0000],[-1,0,-1,0],[9E+09,0.0000,-418.1290,9E+09,9E+09,9E+09]];
	CONST robtarget p611:=[[0.0000,-132.5025,11.6769],[0.0000,-0.1148,-0.9934,0.0000],[-1,0,-1,0],[9E+09,0.0000,-418.9678,9E+09,9E+09,9E+09]];
	CONST robtarget p612:=[[0.0000,-132.9694,11.6962],[0.0000,-0.1220,-0.9925,0.0000],[-1,0,-1,0],[9E+09,0.0000,-419.8008,9E+09,9E+09,9E+09]];
	CONST robtarget p613:=[[0.0000,-133.4642,11.7154],[0.0000,-0.1292,-0.9916,0.0000],[-1,0,-1,0],[9E+09,0.0000,-420.6279,9E+09,9E+09,9E+09]];
	CONST robtarget p614:=[[0.0000,-133.9866,11.7346],[0.0000,-0.1363,-0.9907,0.0000],[-1,0,-1,0],[9E+09,0.0000,-421.4486,9E+09,9E+09,9E+09]];
	CONST robtarget p615:=[[0.0000,-134.5362,11.7538],[0.0000,-0.1433,-0.9897,0.0000],[-1,0,-1,0],[9E+09,0.0000,-422.2628,9E+09,9E+09,9E+09]];
	CONST robtarget p616:=[[0.0000,-135.1128,11.7731],[0.0000,-0.1503,-0.9886,0.0000],[-1,0,-1,0],[9E+09,0.0000,-423.0702,9E+09,9E+09,9E+09]];
	CONST robtarget p617:=[[0.0000,-135.7160,11.7923],[0.0000,-0.1572,-0.9876,0.0000],[-1,0,-1,0],[9E+09,0.0000,-423.8706,9E+09,9E+09,9E+09]];
	CONST robtarget p618:=[[0.0000,-136.3455,11.8115],[0.0000,-0.1640,-0.9865,0.0000],[-1,0,-1,0],[9E+09,0.0000,-424.6638,9E+09,9E+09,9E+09]];
	CONST robtarget p619:=[[0.0000,-137.0008,11.8308],[0.0000,-0.1708,-0.9853,0.0000],[-1,0,-1,0],[9E+09,0.0000,-425.4495,9E+09,9E+09,9E+09]];
	CONST robtarget p620:=[[0.0000,-137.6817,11.8500],[0.0000,-0.1775,-0.9841,0.0000],[-1,0,-1,0],[9E+09,0.0000,-426.2277,9E+09,9E+09,9E+09]];
	CONST robtarget p621:=[[0.0000,-138.3877,11.8692],[0.0000,-0.1841,-0.9829,0.0000],[-1,0,-1,0],[9E+09,0.0000,-426.9980,9E+09,9E+09,9E+09]];
	CONST robtarget p622:=[[0.0000,-139.1184,11.8885],[0.0000,-0.1906,-0.9817,0.0000],[-1,0,-1,0],[9E+09,0.0000,-427.7603,9E+09,9E+09,9E+09]];
	CONST robtarget p623:=[[0.0000,-139.8736,11.9077],[0.0000,-0.1971,-0.9804,0.0000],[-1,0,-1,0],[9E+09,0.0000,-428.5146,9E+09,9E+09,9E+09]];
	CONST robtarget p624:=[[0.0000,-140.6527,11.9269],[0.0000,-0.2034,-0.9791,0.0000],[-1,0,-1,0],[9E+09,0.0000,-429.2606,9E+09,9E+09,9E+09]];
	CONST robtarget p625:=[[0.0000,-141.4553,11.9462],[0.0000,-0.2097,-0.9778,0.0000],[-1,0,-1,0],[9E+09,0.0000,-429.9983,9E+09,9E+09,9E+09]];
	CONST robtarget p626:=[[0.0000,-142.2812,11.9654],[0.0000,-0.2160,-0.9764,0.0000],[-1,0,-1,0],[9E+09,0.0000,-430.7275,9E+09,9E+09,9E+09]];
	CONST robtarget p627:=[[0.0000,-143.1298,11.9846],[0.0000,-0.2221,-0.9750,0.0000],[-1,0,-1,0],[9E+09,0.0000,-431.4482,9E+09,9E+09,9E+09]];
	CONST robtarget p628:=[[0.0000,-144.0009,12.0038],[0.0000,-0.2281,-0.9736,0.0000],[-1,0,-1,0],[9E+09,0.0000,-432.1603,9E+09,9E+09,9E+09]];
	CONST robtarget p629:=[[0.0000,-144.8939,12.0231],[0.0000,-0.2341,-0.9722,0.0000],[-1,0,-1,0],[9E+09,0.0000,-432.8637,9E+09,9E+09,9E+09]];
	CONST robtarget p630:=[[0.0000,-145.8084,12.0423],[0.0000,-0.2400,-0.9708,0.0000],[-1,0,-1,0],[9E+09,0.0000,-433.5584,9E+09,9E+09,9E+09]];
	CONST robtarget p631:=[[0.0000,-146.7442,12.0615],[0.0000,-0.2458,-0.9693,0.0000],[-1,0,-1,0],[9E+09,0.0000,-434.2444,9E+09,9E+09,9E+09]];
	CONST robtarget p632:=[[0.0000,-147.7006,12.0808],[0.0000,-0.2515,-0.9678,0.0000],[-1,0,-1,0],[9E+09,0.0000,-434.9215,9E+09,9E+09,9E+09]];
	CONST robtarget p633:=[[0.0000,-148.6775,12.1000],[0.0000,-0.2572,-0.9664,0.0000],[-1,0,-1,0],[9E+09,0.0000,-435.5899,9E+09,9E+09,9E+09]];
	CONST robtarget p634:=[[0.0000,-149.6743,12.1192],[0.0000,-0.2627,-0.9649,0.0000],[-1,0,-1,0],[9E+09,0.0000,-436.2494,9E+09,9E+09,9E+09]];
	CONST robtarget p635:=[[0.0000,-150.6907,12.1385],[0.0000,-0.2682,-0.9634,0.0000],[-1,0,-1,0],[9E+09,0.0000,-436.9002,9E+09,9E+09,9E+09]];
	CONST robtarget p636:=[[0.0000,-151.7263,12.1577],[0.0000,-0.2736,-0.9618,0.0000],[-1,0,-1,0],[9E+09,0.0000,-437.5421,9E+09,9E+09,9E+09]];
	CONST robtarget p637:=[[0.0000,-152.7806,12.1769],[0.0000,-0.2789,-0.9603,0.0000],[-1,0,-1,0],[9E+09,0.0000,-438.1752,9E+09,9E+09,9E+09]];
	CONST robtarget p638:=[[0.0000,-153.8534,12.1962],[0.0000,-0.2841,-0.9588,0.0000],[-1,0,-1,0],[9E+09,0.0000,-438.7996,9E+09,9E+09,9E+09]];
	CONST robtarget p639:=[[0.0000,-154.9442,12.2154],[0.0000,-0.2893,-0.9572,0.0000],[-1,0,-1,0],[9E+09,0.0000,-439.4153,9E+09,9E+09,9E+09]];
	CONST robtarget p640:=[[0.0000,-156.0526,12.2346],[0.0000,-0.2944,-0.9557,0.0000],[-1,0,-1,0],[9E+09,0.0000,-440.0223,9E+09,9E+09,9E+09]];
	CONST robtarget p641:=[[0.0000,-157.1782,12.2538],[0.0000,-0.2993,-0.9541,0.0000],[-1,0,-1,0],[9E+09,0.0000,-440.6207,9E+09,9E+09,9E+09]];
	CONST robtarget p642:=[[0.0000,-158.3208,12.2731],[0.0000,-0.3042,-0.9526,0.0000],[-1,0,-1,0],[9E+09,0.0000,-441.2104,9E+09,9E+09,9E+09]];
	CONST robtarget p643:=[[0.0000,-159.4799,12.2923],[0.0000,-0.3091,-0.9510,0.0000],[-1,0,-1,0],[9E+09,0.0000,-441.7917,9E+09,9E+09,9E+09]];
	CONST robtarget p644:=[[0.0000,-160.6552,12.3115],[0.0000,-0.3138,-0.9495,0.0000],[-1,0,-1,0],[9E+09,0.0000,-442.3646,9E+09,9E+09,9E+09]];
	CONST robtarget p645:=[[0.0000,-161.8463,12.3308],[0.0000,-0.3185,-0.9479,0.0000],[-1,0,-1,0],[9E+09,0.0000,-442.9290,9E+09,9E+09,9E+09]];
	CONST robtarget p646:=[[0.0000,-163.0529,12.3500],[0.0000,-0.3231,-0.9464,0.0000],[-1,0,-1,0],[9E+09,0.0000,-443.4852,9E+09,9E+09,9E+09]];
	CONST robtarget p647:=[[0.0000,-164.2746,12.3692],[0.0000,-0.3276,-0.9448,0.0000],[-1,0,-1,0],[9E+09,0.0000,-444.0331,9E+09,9E+09,9E+09]];
	CONST robtarget p648:=[[0.0000,-165.5112,12.3885],[0.0000,-0.3321,-0.9433,0.0000],[-1,0,-1,0],[9E+09,0.0000,-444.5729,9E+09,9E+09,9E+09]];
	CONST robtarget p649:=[[0.0000,-166.7622,12.4077],[0.0000,-0.3364,-0.9417,0.0000],[-1,0,-1,0],[9E+09,0.0000,-445.1047,9E+09,9E+09,9E+09]];
	CONST robtarget p650:=[[0.0000,-168.0273,12.4269],[0.0000,-0.3407,-0.9402,0.0000],[-1,0,-1,0],[9E+09,0.0000,-445.6285,9E+09,9E+09,9E+09]];
	CONST robtarget p651:=[[0.0000,-169.3063,12.4462],[0.0000,-0.3450,-0.9386,0.0000],[-1,0,-1,0],[9E+09,0.0000,-446.1444,9E+09,9E+09,9E+09]];
	CONST robtarget p652:=[[0.0000,-170.5988,12.4654],[0.0000,-0.3491,-0.9371,0.0000],[-1,0,-1,0],[9E+09,0.0000,-446.6525,9E+09,9E+09,9E+09]];
	CONST robtarget p653:=[[0.0000,-171.9045,12.4846],[0.0000,-0.3532,-0.9355,0.0000],[-1,0,-1,0],[9E+09,0.0000,-447.1530,9E+09,9E+09,9E+09]];
	CONST robtarget p654:=[[0.0000,-173.2231,12.5038],[0.0000,-0.3572,-0.9340,0.0000],[-1,0,-1,0],[9E+09,0.0000,-447.6458,9E+09,9E+09,9E+09]];
	CONST robtarget p655:=[[0.0000,-174.5544,12.5231],[0.0000,-0.3612,-0.9325,0.0000],[-1,0,-1,0],[9E+09,0.0000,-448.1312,9E+09,9E+09,9E+09]];
	CONST robtarget p656:=[[0.0000,-175.8980,12.5423],[0.0000,-0.3651,-0.9310,0.0000],[-1,0,-1,0],[9E+09,0.0000,-448.6092,9E+09,9E+09,9E+09]];
	CONST robtarget p657:=[[0.0000,-177.2536,12.5615],[0.0000,-0.3689,-0.9295,0.0000],[-1,0,-1,0],[9E+09,0.0000,-449.0800,9E+09,9E+09,9E+09]];
	CONST robtarget p658:=[[0.0000,-178.6211,12.5808],[0.0000,-0.3727,-0.9280,0.0000],[-1,0,-1,0],[9E+09,0.0000,-449.5435,9E+09,9E+09,9E+09]];
	CONST robtarget p659:=[[0.0000,-180.0000,12.6000],[0.0000,-0.3827,0.9239,0.0000],[-1,0,-1,0],[9E+09,0.0000,-450.0000,9E+09,9E+09,9E+09]];
	CONST robtarget p660:=[[0.0000,-178.5993,12.6195],[0.0000,-0.3790,0.9254,0.0000],[-1,0,-1,0],[9E+09,0.0000,-450.4511,9E+09,9E+09,9E+09]];
	CONST robtarget p661:=[[0.0000,-177.2098,12.6391],[0.0000,-0.3753,0.9269,0.0000],[-1,0,-1,0],[9E+09,0.0000,-450.9094,9E+09,9E+09,9E+09]];
	CONST robtarget p662:=[[0.0000,-175.8319,12.6586],[0.0000,-0.3716,0.9284,0.0000],[-1,0,-1,0],[9E+09,0.0000,-451.3748,9E+09,9E+09,9E+09]];
	CONST robtarget p663:=[[0.0000,-174.4657,12.6781],[0.0000,-0.3677,0.9299,0.0000],[-1,0,-1,0],[9E+09,0.0000,-451.8476,9E+09,9E+09,9E+09]];
	CONST robtarget p664:=[[0.0000,-173.1116,12.6977],[0.0000,-0.3638,0.9315,0.0000],[-1,0,-1,0],[9E+09,0.0000,-452.3278,9E+09,9E+09,9E+09]];
	CONST robtarget p665:=[[0.0000,-171.7699,12.7172],[0.0000,-0.3599,0.9330,0.0000],[-1,0,-1,0],[9E+09,0.0000,-452.8156,9E+09,9E+09,9E+09]];
	CONST robtarget p666:=[[0.0000,-170.4407,12.7367],[0.0000,-0.3558,0.9345,0.0000],[-1,0,-1,0],[9E+09,0.0000,-453.3109,9E+09,9E+09,9E+09]];
	CONST robtarget p667:=[[0.0000,-169.1246,12.7562],[0.0000,-0.3517,0.9361,0.0000],[-1,0,-1,0],[9E+09,0.0000,-453.8141,9E+09,9E+09,9E+09]];
	CONST robtarget p668:=[[0.0000,-167.8217,12.7758],[0.0000,-0.3475,0.9377,0.0000],[-1,0,-1,0],[9E+09,0.0000,-454.3251,9E+09,9E+09,9E+09]];
	CONST robtarget p669:=[[0.0000,-166.5323,12.7953],[0.0000,-0.3433,0.9392,0.0000],[-1,0,-1,0],[9E+09,0.0000,-454.8440,9E+09,9E+09,9E+09]];
	CONST robtarget p670:=[[0.0000,-165.2568,12.8148],[0.0000,-0.3390,0.9408,0.0000],[-1,0,-1,0],[9E+09,0.0000,-455.3710,9E+09,9E+09,9E+09]];
	CONST robtarget p671:=[[0.0000,-163.9955,12.8344],[0.0000,-0.3346,0.9424,0.0000],[-1,0,-1,0],[9E+09,0.0000,-455.9061,9E+09,9E+09,9E+09]];
	CONST robtarget p672:=[[0.0000,-162.7488,12.8539],[0.0000,-0.3301,0.9439,0.0000],[-1,0,-1,0],[9E+09,0.0000,-456.4495,9E+09,9E+09,9E+09]];
	CONST robtarget p673:=[[0.0000,-161.5169,12.8734],[0.0000,-0.3256,0.9455,0.0000],[-1,0,-1,0],[9E+09,0.0000,-457.0013,9E+09,9E+09,9E+09]];
	CONST robtarget p674:=[[0.0000,-160.3002,12.8930],[0.0000,-0.3209,0.9471,0.0000],[-1,0,-1,0],[9E+09,0.0000,-457.5614,9E+09,9E+09,9E+09]];
	CONST robtarget p675:=[[0.0000,-159.0990,12.9125],[0.0000,-0.3162,0.9487,0.0000],[-1,0,-1,0],[9E+09,0.0000,-458.1301,9E+09,9E+09,9E+09]];
	CONST robtarget p676:=[[0.0000,-157.9138,12.9320],[0.0000,-0.3114,0.9503,0.0000],[-1,0,-1,0],[9E+09,0.0000,-458.7074,9E+09,9E+09,9E+09]];
	CONST robtarget p677:=[[0.0000,-156.7448,12.9516],[0.0000,-0.3066,0.9518,0.0000],[-1,0,-1,0],[9E+09,0.0000,-459.2933,9E+09,9E+09,9E+09]];
	CONST robtarget p678:=[[0.0000,-155.5925,12.9711],[0.0000,-0.3016,0.9534,0.0000],[-1,0,-1,0],[9E+09,0.0000,-459.8880,9E+09,9E+09,9E+09]];
	CONST robtarget p679:=[[0.0000,-154.4572,12.9906],[0.0000,-0.2966,0.9550,0.0000],[-1,0,-1,0],[9E+09,0.0000,-460.4915,9E+09,9E+09,9E+09]];
	CONST robtarget p680:=[[0.0000,-153.3393,13.0102],[0.0000,-0.2915,0.9566,0.0000],[-1,0,-1,0],[9E+09,0.0000,-461.1038,9E+09,9E+09,9E+09]];
	CONST robtarget p681:=[[0.0000,-152.2391,13.0297],[0.0000,-0.2863,0.9581,0.0000],[-1,0,-1,0],[9E+09,0.0000,-461.7251,9E+09,9E+09,9E+09]];
	CONST robtarget p682:=[[0.0000,-151.1572,13.0492],[0.0000,-0.2810,0.9597,0.0000],[-1,0,-1,0],[9E+09,0.0000,-462.3554,9E+09,9E+09,9E+09]];
	CONST robtarget p683:=[[0.0000,-150.0937,13.0687],[0.0000,-0.2757,0.9612,0.0000],[-1,0,-1,0],[9E+09,0.0000,-462.9946,9E+09,9E+09,9E+09]];
	CONST robtarget p684:=[[0.0000,-149.0492,13.0883],[0.0000,-0.2702,0.9628,0.0000],[-1,0,-1,0],[9E+09,0.0000,-463.6429,9E+09,9E+09,9E+09]];
	CONST robtarget p685:=[[0.0000,-148.0241,13.1078],[0.0000,-0.2647,0.9643,0.0000],[-1,0,-1,0],[9E+09,0.0000,-464.3003,9E+09,9E+09,9E+09]];
	CONST robtarget p686:=[[0.0000,-147.0187,13.1273],[0.0000,-0.2591,0.9659,0.0000],[-1,0,-1,0],[9E+09,0.0000,-464.9667,9E+09,9E+09,9E+09]];
	CONST robtarget p687:=[[0.0000,-146.0335,13.1469],[0.0000,-0.2534,0.9674,0.0000],[-1,0,-1,0],[9E+09,0.0000,-465.6422,9E+09,9E+09,9E+09]];
	CONST robtarget p688:=[[0.0000,-145.0688,13.1664],[0.0000,-0.2476,0.9689,0.0000],[-1,0,-1,0],[9E+09,0.0000,-466.3269,9E+09,9E+09,9E+09]];
	CONST robtarget p689:=[[0.0000,-144.1252,13.1859],[0.0000,-0.2417,0.9703,0.0000],[-1,0,-1,0],[9E+09,0.0000,-467.0205,9E+09,9E+09,9E+09]];
	CONST robtarget p690:=[[0.0000,-143.2029,13.2055],[0.0000,-0.2358,0.9718,0.0000],[-1,0,-1,0],[9E+09,0.0000,-467.7232,9E+09,9E+09,9E+09]];
	CONST robtarget p691:=[[0.0000,-142.3025,13.2250],[0.0000,-0.2298,0.9732,0.0000],[-1,0,-1,0],[9E+09,0.0000,-468.4349,9E+09,9E+09,9E+09]];
	CONST robtarget p692:=[[0.0000,-141.4243,13.2445],[0.0000,-0.2236,0.9747,0.0000],[-1,0,-1,0],[9E+09,0.0000,-469.1556,9E+09,9E+09,9E+09]];
	CONST robtarget p693:=[[0.0000,-140.5687,13.2641],[0.0000,-0.2174,0.9761,0.0000],[-1,0,-1,0],[9E+09,0.0000,-469.8852,9E+09,9E+09,9E+09]];
	CONST robtarget p694:=[[0.0000,-139.7363,13.2836],[0.0000,-0.2111,0.9775,0.0000],[-1,0,-1,0],[9E+09,0.0000,-470.6235,9E+09,9E+09,9E+09]];
	CONST robtarget p695:=[[0.0000,-138.9273,13.3031],[0.0000,-0.2047,0.9788,0.0000],[-1,0,-1,0],[9E+09,0.0000,-471.3706,9E+09,9E+09,9E+09]];
	CONST robtarget p696:=[[0.0000,-138.1421,13.3227],[0.0000,-0.1983,0.9801,0.0000],[-1,0,-1,0],[9E+09,0.0000,-472.1263,9E+09,9E+09,9E+09]];
	CONST robtarget p697:=[[0.0000,-137.3813,13.3422],[0.0000,-0.1917,0.9814,0.0000],[-1,0,-1,0],[9E+09,0.0000,-472.8906,9E+09,9E+09,9E+09]];
	CONST robtarget p698:=[[0.0000,-136.6452,13.3617],[0.0000,-0.1851,0.9827,0.0000],[-1,0,-1,0],[9E+09,0.0000,-473.6631,9E+09,9E+09,9E+09]];
	CONST robtarget p699:=[[0.0000,-135.9343,13.3812],[0.0000,-0.1784,0.9840,0.0000],[-1,0,-1,0],[9E+09,0.0000,-474.4440,9E+09,9E+09,9E+09]];
	CONST robtarget p700:=[[0.0000,-135.2488,13.4008],[0.0000,-0.1716,0.9852,0.0000],[-1,0,-1,0],[9E+09,0.0000,-475.2328,9E+09,9E+09,9E+09]];
	CONST robtarget p701:=[[0.0000,-134.5892,13.4203],[0.0000,-0.1648,0.9863,0.0000],[-1,0,-1,0],[9E+09,0.0000,-476.0296,9E+09,9E+09,9E+09]];
	CONST robtarget p702:=[[0.0000,-133.9559,13.4398],[0.0000,-0.1579,0.9875,0.0000],[-1,0,-1,0],[9E+09,0.0000,-476.8340,9E+09,9E+09,9E+09]];
	CONST robtarget p703:=[[0.0000,-133.3493,13.4594],[0.0000,-0.1509,0.9886,0.0000],[-1,0,-1,0],[9E+09,0.0000,-477.6460,9E+09,9E+09,9E+09]];
	CONST robtarget p704:=[[0.0000,-132.7697,13.4789],[0.0000,-0.1438,0.9896,0.0000],[-1,0,-1,0],[9E+09,0.0000,-478.4652,9E+09,9E+09,9E+09]];
	CONST robtarget p705:=[[0.0000,-132.2174,13.4984],[0.0000,-0.1367,0.9906,0.0000],[-1,0,-1,0],[9E+09,0.0000,-479.2914,9E+09,9E+09,9E+09]];
	CONST robtarget p706:=[[0.0000,-131.6929,13.5180],[0.0000,-0.1295,0.9916,0.0000],[-1,0,-1,0],[9E+09,0.0000,-480.1243,9E+09,9E+09,9E+09]];
	CONST robtarget p707:=[[0.0000,-131.1964,13.5375],[0.0000,-0.1222,0.9925,0.0000],[-1,0,-1,0],[9E+09,0.0000,-480.9638,9E+09,9E+09,9E+09]];
	CONST robtarget p708:=[[0.0000,-130.7283,13.5570],[0.0000,-0.1149,0.9934,0.0000],[-1,0,-1,0],[9E+09,0.0000,-481.8094,9E+09,9E+09,9E+09]];
	CONST robtarget p709:=[[0.0000,-130.2889,13.5766],[0.0000,-0.1075,0.9942,0.0000],[-1,0,-1,0],[9E+09,0.0000,-482.6609,9E+09,9E+09,9E+09]];
	CONST robtarget p710:=[[0.0000,-129.8784,13.5961],[0.0000,-0.1000,0.9950,0.0000],[-1,0,-1,0],[9E+09,0.0000,-483.5180,9E+09,9E+09,9E+09]];
	CONST robtarget p711:=[[0.0000,-129.4972,13.6156],[0.0000,-0.0925,0.9957,0.0000],[-1,0,-1,0],[9E+09,0.0000,-484.3803,9E+09,9E+09,9E+09]];
	CONST robtarget p712:=[[0.0000,-129.1455,13.6352],[0.0000,-0.0850,0.9964,0.0000],[-1,0,-1,0],[9E+09,0.0000,-485.2476,9E+09,9E+09,9E+09]];
	CONST robtarget p713:=[[0.0000,-128.8236,13.6547],[0.0000,-0.0774,0.9970,0.0000],[-1,0,-1,0],[9E+09,0.0000,-486.1193,9E+09,9E+09,9E+09]];
	CONST robtarget p714:=[[0.0000,-128.5316,13.6742],[0.0000,-0.0698,0.9976,0.0000],[-1,0,-1,0],[9E+09,0.0000,-486.9953,9E+09,9E+09,9E+09]];
	CONST robtarget p715:=[[0.0000,-128.2697,13.6937],[0.0000,-0.0621,0.9981,0.0000],[-1,0,-1,0],[9E+09,0.0000,-487.8750,9E+09,9E+09,9E+09]];
	CONST robtarget p716:=[[0.0000,-128.0383,13.7133],[0.0000,-0.0544,0.9985,0.0000],[-1,0,-1,0],[9E+09,0.0000,-488.7581,9E+09,9E+09,9E+09]];
